LIN {X -0.105,Y -512.743,Z 1082.951,A 0.000,B 0.000,C 90.000,E1 27.206} C_DIS
LIN {X -0.246,Y -506.271,Z 1082.947,A 0.000,B 0.000,C 90.000,E1 26.488} C_DIS
LIN {X 0.235,Y -498.378,Z 1082.942,A 0.000,B 0.000,C 90.000,E1 25.591} C_DIS
LIN {X 0.081,Y -491.474,Z 1082.938,A 0.000,B 0.000,C 90.000,E1 24.899} C_DIS
LIN {X 0.101,Y -483.056,Z 1082.934,A 0.000,B 0.000,C 90.000,E1 24.079} C_DIS
LIN {X 0.080,Y -473.077,Z 1082.929,A 0.000,B 0.000,C 90.000,E1 23.153} C_DIS
LIN {X -0.074,Y -468.531,Z 1082.927,A 0.000,B 0.000,C 90.000,E1 22.770} C_DIS
LIN {X 0.200,Y -458.259,Z 1082.922,A 0.000,B 0.000,C 90.000,E1 21.844} C_DIS
LIN {X -0.133,Y -450.699,Z 1082.918,A 0.000,B 0.000,C 90.000,E1 21.227} C_DIS
LIN {X -0.068,Y -433.276,Z 1082.909,A 0.000,B 0.000,C 90.000,E1 19.631} C_DIS
LIN {X -0.013,Y -417.456,Z 1082.900,A 0.000,B 0.000,C 90.000,E1 18.000} C_DIS
LIN {X 0.024,Y -405.312,Z 1082.892,A 0.000,B 0.000,C 90.000,E1 16.567} C_DIS
LIN {X 0.104,Y -399.058,Z 1082.887,A 0.000,B 0.000,C 90.000,E1 15.717} C_DIS
LIN {X 0.077,Y -396.824,Z 1082.885,A 0.000,B 0.000,C 90.000,E1 15.371} C_DIS
LIN {X -0.054,Y -394.256,Z 1082.883,A 0.000,B 0.000,C 90.000,E1 14.898} C_DIS
LIN {X 0.015,Y -392.680,Z 1082.880,A 0.000,B 0.000,C 90.000,E1 14.356} C_DIS
LIN {X -0.009,Y -392.087,Z 1082.877,A 0.000,B 0.000,C 90.000,E1 13.828} C_DIS
LIN {X 0.012,Y -392.010,Z 1082.876,A 0.000,B 0.000,C 90.000,E1 13.647} C_DIS
LIN {X -0.076,Y -392.528,Z 1082.871,A 0.000,B 0.000,C 90.000,E1 12.771} C_DIS
LIN {X -0.071,Y -394.325,Z 1082.863,A 0.000,B 0.000,C 90.000,E1 11.366} C_DIS
LIN {X 0.118,Y -400.821,Z 1082.844,A 0.000,B 0.000,C 90.000,E1 7.814} C_DIS
LIN {X -0.026,Y -405.485,Z 1082.832,A 0.000,B 0.000,C 90.000,E1 5.739} C_DIS
LIN {X -0.062,Y -406.947,Z 1082.828,A 0.000,B 0.000,C 90.000,E1 5.049} C_DIS
LIN {X -0.086,Y -409.086,Z 1082.824,A 0.000,B 0.000,C 90.000,E1 4.359} C_DIS
LIN {X -0.078,Y -410.586,Z 1082.822,A 0.000,B 0.000,C 90.000,E1 4.012} C_DIS
LIN {X -0.092,Y -412.395,Z 1082.820,A 0.000,B 0.000,C 90.000,E1 3.669} C_DIS
LIN {X -0.098,Y -415.251,Z 1082.818,A 0.000,B 0.000,C 90.000,E1 3.326} C_DIS
LIN {X 0.044,Y -417.972,Z 1082.817,A 0.000,B 0.000,C 90.000,E1 3.037} C_DIS
LIN {X 0.077,Y -421.563,Z 1082.815,A 0.000,B 0.000,C 90.000,E1 2.751} C_DIS
LIN {X -0.121,Y -429.063,Z 1082.813,A 0.000,B 0.000,C 90.000,E1 2.293} C_DIS
LIN {X 0.017,Y -448.904,Z 1082.805,A 0.000,B 0.000,C 90.000,E1 0.974} C_DIS
LIN {X 0.000,Y -464.386,Z 1082.800,A 0.000,B 0.000,C 90.000,E1 360.000} C_DIS
LIN {X 0.157,Y -474.218,Z 1082.797,A 0.000,B 0.000,C 90.000,E1 359.370} C_DIS
LIN {X -0.054,Y -485.618,Z 1082.793,A 0.000,B 0.000,C 90.000,E1 358.682} C_DIS
LIN {X -0.189,Y -491.941,Z 1082.790,A 0.000,B 0.000,C 90.000,E1 358.282} C_DIS
LIN {X 0.157,Y -499.792,Z 1082.787,A 0.000,B 0.000,C 90.000,E1 357.707} C_DIS
LIN {X -0.201,Y -504.418,Z 1082.786,A 0.000,B 0.000,C 90.000,E1 357.421} C_DIS
LIN {X -0.122,Y -510.460,Z 1082.783,A 0.000,B 0.000,C 90.000,E1 356.963} C_DIS
LIN {X -0.140,Y -516.466,Z 1082.781,A 0.000,B 0.000,C 90.000,E1 356.502} C_DIS
LIN {X 0.074,Y -523.648,Z 1082.777,A 0.000,B 0.000,C 90.000,E1 355.869} C_DIS
LIN {X 0.106,Y -528.999,Z 1082.774,A 0.000,B 0.000,C 90.000,E1 355.355} C_DIS
LIN {X -0.259,Y -533.999,Z 1082.771,A 0.000,B 0.000,C 90.000,E1 354.894} C_DIS
LIN {X -0.088,Y -539.075,Z 1082.768,A 0.000,B 0.000,C 90.000,E1 354.318} C_DIS
LIN {X 0.248,Y -544.958,Z 1082.765,A 0.000,B 0.000,C 90.000,E1 353.571} C_DIS
LIN {X 0.066,Y -548.338,Z 1082.762,A 0.000,B 0.000,C 90.000,E1 353.166} C_DIS
LIN {X 0.008,Y -553.208,Z 1082.758,A 0.000,B 0.000,C 90.000,E1 352.470} C_DIS
LIN {X -0.083,Y -557.570,Z 1082.754,A 0.000,B 0.000,C 90.000,E1 351.781} C_DIS
LIN {X 0.189,Y -560.730,Z 1082.751,A 0.000,B 0.000,C 90.000,E1 351.197} C_DIS
LIN {X 0.248,Y -564.312,Z 1082.747,A 0.000,B 0.000,C 90.000,E1 350.500} C_DIS
LIN {X -0.221,Y -567.611,Z 1082.744,A 0.000,B 0.000,C 90.000,E1 349.859} C_DIS
LIN {X 0.031,Y -570.045,Z 1082.741,A 0.000,B 0.000,C 90.000,E1 349.285} C_DIS
LIN {X 0.226,Y -574.569,Z 1082.734,A 0.000,B 0.000,C 90.000,E1 348.173} C_DIS
LIN {X -0.288,Y -577.679,Z 1082.730,A 0.000,B 0.000,C 90.000,E1 347.409} C_DIS
LIN {X -0.208,Y -580.742,Z 1082.725,A 0.000,B 0.000,C 90.000,E1 346.589} C_DIS
LIN {X 0.182,Y -586.351,Z 1082.716,A 0.000,B 0.000,C 90.000,E1 344.936} C_DIS
LIN {X 0.028,Y -590.694,Z 1082.709,A 0.000,B 0.000,C 90.000,E1 343.614} C_DIS
LIN {X -0.219,Y -594.814,Z 1082.702,A 0.000,B 0.000,C 90.000,E1 342.308} C_DIS
LIN {X 0.070,Y -598.009,Z 1082.696,A 0.000,B 0.000,C 90.000,E1 341.221} C_DIS
LIN {X 0.019,Y -602.177,Z 1082.687,A 0.000,B 0.000,C 90.000,E1 339.645} C_DIS
LIN {X 0.127,Y -604.055,Z 1082.683,A 0.000,B 0.000,C 90.000,E1 338.847} C_DIS
LIN {X 0.191,Y -606.370,Z 1082.677,A 0.000,B 0.000,C 90.000,E1 337.794} C_DIS
LIN {X 0.236,Y -608.760,Z 1082.670,A 0.000,B 0.000,C 90.000,E1 336.485} C_DIS
LIN {X -0.194,Y -610.357,Z 1082.664,A 0.000,B 0.000,C 90.000,E1 335.485} C_DIS
LIN {X 0.240,Y -611.498,Z 1082.659,A 0.000,B 0.000,C 90.000,E1 334.665} C_DIS
LIN {X 0.073,Y -613.069,Z 1082.652,A 0.000,B 0.000,C 90.000,E1 333.384} C_DIS
LIN {X -0.015,Y -613.870,Z 1082.648,A 0.000,B 0.000,C 90.000,E1 332.615} C_DIS
LIN {X 0.168,Y -614.764,Z 1082.642,A 0.000,B 0.000,C 90.000,E1 331.563} C_DIS
LIN {X 0.066,Y -615.301,Z 1082.636,A 0.000,B 0.000,C 90.000,E1 330.539} C_DIS
LIN {X -0.268,Y -615.607,Z 1082.631,A 0.000,B 0.000,C 90.000,E1 329.537} C_DIS
LIN {X 0.252,Y -615.430,Z 1082.625,A 0.000,B 0.000,C 90.000,E1 328.456} C_DIS
LIN {X -0.077,Y -614.933,Z 1082.619,A 0.000,B 0.000,C 90.000,E1 327.454} C_DIS
LIN {X -0.085,Y -614.033,Z 1082.613,A 0.000,B 0.000,C 90.000,E1 326.421} C_DIS
LIN {X 0.189,Y -612.460,Z 1082.606,A 0.000,B 0.000,C 90.000,E1 325.102} C_DIS
LIN {X -0.146,Y -611.447,Z 1082.602,A 0.000,B 0.000,C 90.000,E1 324.356} C_DIS
LIN {X 0.224,Y -609.559,Z 1082.593,A 0.000,B 0.000,C 90.000,E1 322.763} C_DIS
LIN {X -0.293,Y -607.736,Z 1082.585,A 0.000,B 0.000,C 90.000,E1 321.251} C_DIS
LIN {X -0.082,Y -606.156,Z 1082.576,A 0.000,B 0.000,C 90.000,E1 319.666} C_DIS
LIN {X -0.097,Y -604.273,Z 1082.566,A 0.000,B 0.000,C 90.000,E1 317.838} C_DIS
LIN {X -0.049,Y -603.668,Z 1082.563,A 0.000,B 0.000,C 90.000,E1 317.310} C_DIS
LIN {X -0.209,Y -602.585,Z 1082.558,A 0.000,B 0.000,C 90.000,E1 316.539} C_DIS
LIN {X 0.060,Y -599.970,Z 1082.548,A 0.000,B 0.000,C 90.000,E1 314.676} C_DIS
LIN {X -0.152,Y -598.236,Z 1082.541,A 0.000,B 0.000,C 90.000,E1 313.380} C_DIS
LIN {X 0.246,Y -595.387,Z 1082.529,A 0.000,B 0.000,C 90.000,E1 311.229} C_DIS
LIN {X -0.018,Y -593.384,Z 1082.522,A 0.000,B 0.000,C 90.000,E1 309.930} C_DIS
LIN {X 0.169,Y -592.012,Z 1082.517,A 0.000,B 0.000,C 90.000,E1 309.116} C_DIS
LIN {X -0.074,Y -589.339,Z 1082.510,A 0.000,B 0.000,C 90.000,E1 307.810} C_DIS
LIN {X 0.108,Y -586.240,Z 1082.503,A 0.000,B 0.000,C 90.000,E1 306.457} C_DIS
LIN {X 0.020,Y -584.738,Z 1082.500,A 0.000,B 0.000,C 90.000,E1 305.931} C_DIS
LIN {X -0.134,Y -583.880,Z 1082.498,A 0.000,B 0.000,C 90.000,E1 305.678} C_DIS
LIN {X 0.233,Y -582.438,Z 1082.495,A 0.000,B 0.000,C 90.000,E1 305.105} C_DIS
LIN {X -0.223,Y -580.788,Z 1082.492,A 0.000,B 0.000,C 90.000,E1 304.612} C_DIS
LIN {X 0.115,Y -578.836,Z 1082.489,A 0.000,B 0.000,C 90.000,E1 304.040} C_DIS
LIN {X 0.114,Y -576.720,Z 1082.486,A 0.000,B 0.000,C 90.000,E1 303.499} C_DIS
LIN {X 0.013,Y -573.478,Z 1082.482,A 0.000,B 0.000,C 90.000,E1 302.832} C_DIS
LIN {X 0.013,Y -568.208,Z 1082.477,A 0.000,B 0.000,C 90.000,E1 301.878} C_DIS
LIN {X -0.079,Y -567.363,Z 1082.476,A 0.000,B 0.000,C 90.000,E1 301.750} C_DIS
LIN {X -0.063,Y -560.691,Z 1082.472,A 0.000,B 0.000,C 90.000,E1 300.924} C_DIS
LIN {X -0.157,Y -555.536,Z 1082.469,A 0.000,B 0.000,C 90.000,E1 300.384} C_DIS
LIN {X -0.123,Y -552.525,Z 1082.467,A 0.000,B 0.000,C 90.000,E1 300.129} C_DIS
LIN {X 0.055,Y -547.457,Z 1082.465,A 0.000,B 0.000,C 90.000,E1 299.617} C_DIS
LIN {X -0.277,Y -546.455,Z 1082.464,A 0.000,B 0.000,C 90.000,E1 299.539} C_DIS
LIN {X -0.028,Y -544.583,Z 1082.462,A 0.000,B 0.000,C 90.000,E1 299.205} C_DIS
LIN {X -0.152,Y -543.636,Z 1082.462,A 0.000,B 0.000,C 90.000,E1 299.077} C_DIS
LIN {X 0.205,Y -542.356,Z 1082.459,A 0.000,B 0.000,C 90.000,E1 298.615} C_DIS
LIN {X 0.076,Y -542.284,Z 1082.458,A 0.000,B 0.000,C 90.000,E1 298.487} C_DIS
LIN {X -0.150,Y -542.015,Z 1082.458,A 0.000,B 0.000,C 90.000,E1 298.359} C_DIS
LIN {X 0.069,Y -541.254,Z 1082.456,A 0.000,B 0.000,C 90.000,E1 298.052} C_DIS
LIN {X 0.063,Y -541.031,Z 1082.454,A 0.000,B 0.000,C 90.000,E1 297.769} C_DIS
LIN {X 0.149,Y -540.497,Z 1082.452,A 0.000,B 0.000,C 90.000,E1 297.334} C_DIS
LIN {X 0.019,Y -540.575,Z 1082.451,A 0.000,B 0.000,C 90.000,E1 297.206} C_DIS
LIN {X 0.000,Y -540.494,Z 1082.450,A 0.000,B 0.000,C 90.000,E1 296.924} C_DIS
LIN {X 0.219,Y -540.223,Z 1082.448,A 0.000,B 0.000,C 90.000,E1 296.616} C_DIS
LIN {X 0.061,Y -540.481,Z 1082.431,A 0.000,B 0.000,C 90.000,E1 293.590} C_DIS
LIN {X 0.215,Y -540.875,Z 1082.423,A 0.000,B 0.000,C 90.000,E1 292.153} C_DIS
LIN {X -0.105,Y -541.428,Z 1082.414,A 0.000,B 0.000,C 90.000,E1 290.482} C_DIS
LIN {X 0.126,Y -541.613,Z 1082.407,A 0.000,B 0.000,C 90.000,E1 289.322} C_DIS
LIN {X 0.183,Y -541.648,Z 1082.401,A 0.000,B 0.000,C 90.000,E1 288.181} C_DIS
LIN {X 0.015,Y -541.453,Z 1082.392,A 0.000,B 0.000,C 90.000,E1 286.496} C_DIS
LIN {X 0.134,Y -541.076,Z 1082.384,A 0.000,B 0.000,C 90.000,E1 285.064} C_DIS
LIN {X 0.104,Y -540.565,Z 1082.376,A 0.000,B 0.000,C 90.000,E1 283.647} C_DIS
LIN {X -0.055,Y -539.946,Z 1082.368,A 0.000,B 0.000,C 90.000,E1 282.243} C_DIS
LIN {X -0.219,Y -539.205,Z 1082.360,A 0.000,B 0.000,C 90.000,E1 280.838} C_DIS
LIN {X 0.233,Y -538.052,Z 1082.347,A 0.000,B 0.000,C 90.000,E1 278.511} C_DIS
LIN {X -0.089,Y -537.157,Z 1082.338,A 0.000,B 0.000,C 90.000,E1 276.834} C_DIS
LIN {X 0.042,Y -536.295,Z 1082.328,A 0.000,B 0.000,C 90.000,E1 275.106} C_DIS
LIN {X 0.112,Y -535.382,Z 1082.319,A 0.000,B 0.000,C 90.000,E1 273.383} C_DIS
LIN {X 0.154,Y -534.529,Z 1082.309,A 0.000,B 0.000,C 90.000,E1 271.661} C_DIS
LIN {X 0.147,Y -534.032,Z 1082.303,A 0.000,B 0.000,C 90.000,E1 270.516} C_DIS
LIN {X 0.126,Y -533.069,Z 1082.293,A 0.000,B 0.000,C 90.000,E1 268.797} C_DIS
LIN {X 0.092,Y -532.058,Z 1082.284,A 0.000,B 0.000,C 90.000,E1 267.078} C_DIS
LIN {X 0.100,Y -531.420,Z 1082.277,A 0.000,B 0.000,C 90.000,E1 265.927} C_DIS
LIN {X 0.058,Y -530.119,Z 1082.268,A 0.000,B 0.000,C 90.000,E1 264.204} C_DIS
LIN {X 0.066,Y -528.841,Z 1082.260,A 0.000,B 0.000,C 90.000,E1 262.761} C_DIS
LIN {X 0.093,Y -526.698,Z 1082.249,A 0.000,B 0.000,C 90.000,E1 260.735} C_DIS
LIN {X 0.107,Y -525.157,Z 1082.241,A 0.000,B 0.000,C 90.000,E1 259.285} C_DIS
LIN {X 0.184,Y -523.654,Z 1082.233,A 0.000,B 0.000,C 90.000,E1 257.825} C_DIS
LIN {X -0.156,Y -521.929,Z 1082.223,A 0.000,B 0.000,C 90.000,E1 256.117} C_DIS
LIN {X 0.104,Y -520.178,Z 1082.213,A 0.000,B 0.000,C 90.000,E1 254.338} C_DIS
LIN {X -0.029,Y -518.351,Z 1082.203,A 0.000,B 0.000,C 90.000,E1 252.598} C_DIS
LIN {X -0.167,Y -516.791,Z 1082.195,A 0.000,B 0.000,C 90.000,E1 251.148} C_DIS
LIN {X 0.143,Y -515.178,Z 1082.187,A 0.000,B 0.000,C 90.000,E1 249.645} C_DIS
LIN {X -0.057,Y -512.961,Z 1082.177,A 0.000,B 0.000,C 90.000,E1 247.901} C_DIS
LIN {X 0.180,Y -510.485,Z 1082.167,A 0.000,B 0.000,C 90.000,E1 246.102} C_DIS
LIN {X 0.141,Y -508.671,Z 1082.161,A 0.000,B 0.000,C 90.000,E1 244.921} C_DIS
LIN {X -0.173,Y -506.824,Z 1082.154,A 0.000,B 0.000,C 90.000,E1 243.768} C_DIS
LIN {X -0.139,Y -505.365,Z 1082.149,A 0.000,B 0.000,C 90.000,E1 242.871} C_DIS
LIN {X -0.193,Y -502.859,Z 1082.141,A 0.000,B 0.000,C 90.000,E1 241.385} C_DIS
LIN {X 0.237,Y -499.776,Z 1082.131,A 0.000,B 0.000,C 90.000,E1 239.537} C_DIS
LIN {X -0.257,Y -496.507,Z 1082.121,A 0.000,B 0.000,C 90.000,E1 237.788} C_DIS
LIN {X 0.131,Y -493.104,Z 1082.111,A 0.000,B 0.000,C 90.000,E1 235.928} C_DIS
LIN {X 0.189,Y -490.141,Z 1082.102,A 0.000,B 0.000,C 90.000,E1 234.402} C_DIS
LIN {X -0.213,Y -487.095,Z 1082.094,A 0.000,B 0.000,C 90.000,E1 232.924} C_DIS
LIN {X 0.118,Y -483.221,Z 1082.084,A 0.000,B 0.000,C 90.000,E1 231.045} C_DIS
LIN {X -0.200,Y -479.911,Z 1082.075,A 0.000,B 0.000,C 90.000,E1 229.542} C_DIS
LIN {X 0.094,Y -474.844,Z 1082.061,A 0.000,B 0.000,C 90.000,E1 227.025} C_DIS
LIN {X 0.103,Y -470.752,Z 1082.049,A 0.000,B 0.000,C 90.000,E1 224.838} C_DIS
LIN {X -0.070,Y -467.249,Z 1082.039,A 0.000,B 0.000,C 90.000,E1 222.975} C_DIS
LIN {X 0.166,Y -465.471,Z 1082.033,A 0.000,B 0.000,C 90.000,E1 222.000} C_DIS
LIN {X -0.017,Y -461.185,Z 1082.021,A 0.000,B 0.000,C 90.000,E1 219.806} C_DIS
LIN {X -0.082,Y -458.171,Z 1082.012,A 0.000,B 0.000,C 90.000,E1 218.222} C_DIS
LIN {X -0.048,Y -454.475,Z 1082.002,A 0.000,B 0.000,C 90.000,E1 216.297} C_DIS
LIN {X -0.159,Y -452.026,Z 1081.995,A 0.000,B 0.000,C 90.000,E1 215.025} C_DIS
LIN {X -0.005,Y -447.147,Z 1081.980,A 0.000,B 0.000,C 90.000,E1 212.418} C_DIS
LIN {X 0.018,Y -443.605,Z 1081.969,A 0.000,B 0.000,C 90.000,E1 210.463} C_DIS
LIN {X 0.112,Y -440.141,Z 1081.958,A 0.000,B 0.000,C 90.000,E1 208.487} C_DIS
LIN {X 0.148,Y -435.672,Z 1081.944,A 0.000,B 0.000,C 90.000,E1 205.848} C_DIS
LIN {X 0.214,Y -433.861,Z 1081.936,A 0.000,B 0.000,C 90.000,E1 204.515} C_DIS
LIN {X -0.099,Y -430.329,Z 1081.922,A 0.000,B 0.000,C 90.000,E1 201.897} C_DIS
LIN {X -0.243,Y -428.987,Z 1081.912,A 0.000,B 0.000,C 90.000,E1 200.248} C_DIS
LIN {X -0.227,Y -428.850,Z 1081.909,A 0.000,B 0.000,C 90.000,E1 199.577} C_DIS
LIN {X -0.213,Y -429.007,Z 1081.905,A 0.000,B 0.000,C 90.000,E1 198.906} C_DIS
LIN {X 0.207,Y -429.520,Z 1081.901,A 0.000,B 0.000,C 90.000,E1 198.181} C_DIS
LIN {X 0.221,Y -430.422,Z 1081.897,A 0.000,B 0.000,C 90.000,E1 197.511} C_DIS
LIN {X 0.111,Y -431.796,Z 1081.894,A 0.000,B 0.000,C 90.000,E1 196.858} C_DIS
LIN {X -0.085,Y -432.640,Z 1081.892,A 0.000,B 0.000,C 90.000,E1 196.551} C_DIS
LIN {X -0.069,Y -435.929,Z 1081.886,A 0.000,B 0.000,C 90.000,E1 195.552} C_DIS
LIN {X 0.107,Y -443.669,Z 1081.876,A 0.000,B 0.000,C 90.000,E1 193.716} C_DIS
LIN {X 0.166,Y -450.524,Z 1081.868,A 0.000,B 0.000,C 90.000,E1 192.243} C_DIS
LIN {X -0.068,Y -457.822,Z 1081.860,A 0.000,B 0.000,C 90.000,E1 190.838} C_DIS
LIN {X 0.113,Y -467.048,Z 1081.851,A 0.000,B 0.000,C 90.000,E1 189.095} C_DIS
LIN {X 0.063,Y -475.533,Z 1081.842,A 0.000,B 0.000,C 90.000,E1 187.530} C_DIS
LIN {X -0.011,Y -480.533,Z 1081.837,A 0.000,B 0.000,C 90.000,E1 186.606} C_DIS
LIN {X 0.116,Y -486.113,Z 1081.831,A 0.000,B 0.000,C 90.000,E1 185.511} C_DIS
LIN {X -0.009,Y -492.414,Z 1081.824,A 0.000,B 0.000,C 90.000,E1 184.302} C_DIS
LIN {X 0.129,Y -499.320,Z 1081.816,A 0.000,B 0.000,C 90.000,E1 182.922} C_DIS
LIN {X -0.053,Y -504.614,Z 1081.811,A 0.000,B 0.000,C 90.000,E1 181.892} C_DIS
LIN {X -0.244,Y -511.387,Z 1081.803,A 0.000,B 0.000,C 90.000,E1 180.573} C_DIS
LIN {X -0.170,Y -520.402,Z 1081.793,A 0.000,B 0.000,C 90.000,E1 178.797} C_DIS
LIN {X 0.145,Y -527.773,Z 1081.785,A 0.000,B 0.000,C 90.000,E1 177.306} C_DIS
LIN {X -0.194,Y -534.352,Z 1081.778,A 0.000,B 0.000,C 90.000,E1 176.045} C_DIS
LIN {X -0.124,Y -541.601,Z 1081.770,A 0.000,B 0.000,C 90.000,E1 174.609} C_DIS
LIN {X 0.110,Y -547.347,Z 1081.764,A 0.000,B 0.000,C 90.000,E1 173.451} C_DIS
LIN {X -0.017,Y -555.815,Z 1081.754,A 0.000,B 0.000,C 90.000,E1 171.781} C_DIS
LIN {X 0.281,Y -561.957,Z 1081.747,A 0.000,B 0.000,C 90.000,E1 170.500} C_DIS
LIN {X -0.110,Y -568.683,Z 1081.740,A 0.000,B 0.000,C 90.000,E1 169.162} C_DIS
LIN {X 0.282,Y -575.057,Z 1081.732,A 0.000,B 0.000,C 90.000,E1 167.757} C_DIS
LIN {X -0.017,Y -581.736,Z 1081.724,A 0.000,B 0.000,C 90.000,E1 166.297} C_DIS
LIN {X -0.168,Y -587.013,Z 1081.717,A 0.000,B 0.000,C 90.000,E1 165.102} C_DIS
LIN {X 0.102,Y -592.400,Z 1081.710,A 0.000,B 0.000,C 90.000,E1 163.740} C_DIS
LIN {X -0.081,Y -595.449,Z 1081.705,A 0.000,B 0.000,C 90.000,E1 162.960} C_DIS
LIN {X 0.224,Y -599.333,Z 1081.699,A 0.000,B 0.000,C 90.000,E1 161.873} C_DIS
LIN {X 0.111,Y -602.132,Z 1081.695,A 0.000,B 0.000,C 90.000,E1 161.094} C_DIS
LIN {X -0.135,Y -606.421,Z 1081.688,A 0.000,B 0.000,C 90.000,E1 159.806} C_DIS
LIN {X 0.265,Y -610.476,Z 1081.681,A 0.000,B 0.000,C 90.000,E1 158.465} C_DIS
LIN {X 0.154,Y -614.298,Z 1081.673,A 0.000,B 0.000,C 90.000,E1 157.177} C_DIS
LIN {X -0.227,Y -617.908,Z 1081.666,A 0.000,B 0.000,C 90.000,E1 155.921} C_DIS
LIN {X 0.006,Y -621.912,Z 1081.658,A 0.000,B 0.000,C 90.000,E1 154.357} C_DIS
LIN {X 0.013,Y -625.143,Z 1081.651,A 0.000,B 0.000,C 90.000,E1 153.076} C_DIS
LIN {X 0.368,Y -628.222,Z 1081.643,A 0.000,B 0.000,C 90.000,E1 151.769} C_DIS
LIN {X -0.076,Y -631.141,Z 1081.636,A 0.000,B 0.000,C 90.000,E1 150.539} C_DIS
LIN {X 0.187,Y -634.472,Z 1081.628,A 0.000,B 0.000,C 90.000,E1 148.997} C_DIS
LIN {X -0.013,Y -637.709,Z 1081.620,A 0.000,B 0.000,C 90.000,E1 147.502} C_DIS
LIN {X -0.114,Y -641.275,Z 1081.610,A 0.000,B 0.000,C 90.000,E1 145.754} C_DIS
LIN {X 0.048,Y -644.710,Z 1081.600,A 0.000,B 0.000,C 90.000,E1 143.989} C_DIS
LIN {X 0.252,Y -647.511,Z 1081.592,A 0.000,B 0.000,C 90.000,E1 142.477} C_DIS
LIN {X 0.078,Y -649.950,Z 1081.585,A 0.000,B 0.000,C 90.000,E1 141.251} C_DIS
LIN {X -0.187,Y -653.393,Z 1081.575,A 0.000,B 0.000,C 90.000,E1 139.542} C_DIS
LIN {X 0.088,Y -656.414,Z 1081.567,A 0.000,B 0.000,C 90.000,E1 138.038} C_DIS
LIN {X 0.306,Y -661.064,Z 1081.555,A 0.000,B 0.000,C 90.000,E1 135.810} C_DIS
LIN {X 0.215,Y -665.116,Z 1081.545,A 0.000,B 0.000,C 90.000,E1 134.109} C_DIS
LIN {X -0.248,Y -670.050,Z 1081.534,A 0.000,B 0.000,C 90.000,E1 132.204} C_DIS
LIN {X 0.385,Y -674.371,Z 1081.525,A 0.000,B 0.000,C 90.000,E1 130.458} C_DIS
LIN {X 0.140,Y -678.018,Z 1081.517,A 0.000,B 0.000,C 90.000,E1 129.036} C_DIS
LIN {X -0.293,Y -682.977,Z 1081.506,A 0.000,B 0.000,C 90.000,E1 127.156} C_DIS
LIN {X 0.113,Y -686.067,Z 1081.500,A 0.000,B 0.000,C 90.000,E1 125.931} C_DIS
LIN {X -0.204,Y -689.531,Z 1081.492,A 0.000,B 0.000,C 90.000,E1 124.532} C_DIS
LIN {X -0.241,Y -693.558,Z 1081.483,A 0.000,B 0.000,C 90.000,E1 122.880} C_DIS
LIN {X -0.218,Y -696.953,Z 1081.475,A 0.000,B 0.000,C 90.000,E1 121.465} C_DIS
LIN {X -0.050,Y -699.009,Z 1081.469,A 0.000,B 0.000,C 90.000,E1 120.512} C_DIS
LIN {X 0.128,Y -700.324,Z 1081.466,A 0.000,B 0.000,C 90.000,E1 119.795} C_DIS
LIN {X 0.053,Y -701.043,Z 1081.463,A 0.000,B 0.000,C 90.000,E1 119.333} C_DIS
LIN {X 0.188,Y -702.361,Z 1081.457,A 0.000,B 0.000,C 90.000,E1 118.153} C_DIS
LIN {X 0.298,Y -703.666,Z 1081.449,A 0.000,B 0.000,C 90.000,E1 116.744} C_DIS
LIN {X 0.149,Y -704.730,Z 1081.442,A 0.000,B 0.000,C 90.000,E1 115.591} C_DIS
LIN {X -0.216,Y -705.058,Z 1081.440,A 0.000,B 0.000,C 90.000,E1 115.155} C_DIS
LIN {X 0.360,Y -705.140,Z 1081.437,A 0.000,B 0.000,C 90.000,E1 114.643} C_DIS
LIN {X 0.002,Y -704.721,Z 1081.435,A 0.000,B 0.000,C 90.000,E1 114.207} C_DIS
LIN {X 0.287,Y -704.411,Z 1081.433,A 0.000,B 0.000,C 90.000,E1 113.951} C_DIS
LIN {X -0.074,Y -702.806,Z 1081.431,A 0.000,B 0.000,C 90.000,E1 113.515} C_DIS
LIN {X 0.204,Y -701.746,Z 1081.429,A 0.000,B 0.000,C 90.000,E1 113.259} C_DIS
LIN {X -0.173,Y -698.154,Z 1081.427,A 0.000,B 0.000,C 90.000,E1 112.823} C_DIS
LIN {X -0.044,Y -697.056,Z 1081.426,A 0.000,B 0.000,C 90.000,E1 112.695} C_DIS
LIN {X -0.182,Y -695.384,Z 1081.425,A 0.000,B 0.000,C 90.000,E1 112.589} C_DIS
LIN {X 0.363,Y -687.730,Z 1081.424,A 0.000,B 0.000,C 90.000,E1 112.206} C_DIS
LIN {X 0.141,Y -685.814,Z 1081.423,A 0.000,B 0.000,C 90.000,E1 112.153} C_DIS
LIN {X -0.285,Y -684.330,Z 1081.423,A 0.000,B 0.000,C 90.000,E1 112.153} C_DIS
LIN {X -0.082,Y -675.933,Z 1081.422,A 0.000,B 0.000,C 90.000,E1 112.025} C_DIS
LIN {X -0.121,Y -605.703,Z 1081.422,A 0.000,B 0.000,C 90.000,E1 112.025} C_DIS
LIN {X -0.017,Y -601.930,Z 1081.421,A 0.000,B 0.000,C 90.000,E1 111.844} C_DIS
LIN {X 0.141,Y -596.452,Z 1081.419,A 0.000,B 0.000,C 90.000,E1 111.482} C_DIS
LIN {X 0.237,Y -587.291,Z 1081.415,A 0.000,B 0.000,C 90.000,E1 110.737} C_DIS
LIN {X -0.108,Y -578.950,Z 1081.411,A 0.000,B 0.000,C 90.000,E1 110.066} C_DIS
LIN {X 0.022,Y -574.660,Z 1081.410,A 0.000,B 0.000,C 90.000,E1 109.704} C_DIS
LIN {X -0.127,Y -568.620,Z 1081.407,A 0.000,B 0.000,C 90.000,E1 109.268} C_DIS
LIN {X 0.186,Y -560.275,Z 1081.404,A 0.000,B 0.000,C 90.000,E1 108.725} C_DIS
LIN {X 0.113,Y -553.840,Z 1081.402,A 0.000,B 0.000,C 90.000,E1 108.362} C_DIS
LIN {X 0.190,Y -549.451,Z 1081.401,A 0.000,B 0.000,C 90.000,E1 108.055} C_DIS
LIN {X -0.059,Y -547.800,Z 1081.399,A 0.000,B 0.000,C 90.000,E1 107.873} C_DIS
LIN {X -0.090,Y -547.793,Z 1081.399,A 0.000,B 0.000,C 90.000,E1 107.873} C_DIS
LIN {X -0.214,Y -547.542,Z 1081.398,A 0.000,B 0.000,C 90.000,E1 107.692} C_DIS
LIN {X 0.214,Y -547.463,Z 1081.397,A 0.000,B 0.000,C 90.000,E1 107.457} C_DIS
LIN {X 0.053,Y -548.752,Z 1081.385,A 0.000,B 0.000,C 90.000,E1 105.300} C_DIS
LIN {X -0.155,Y -550.211,Z 1081.374,A 0.000,B 0.000,C 90.000,E1 103.355} C_DIS
LIN {X -0.132,Y -551.386,Z 1081.366,A 0.000,B 0.000,C 90.000,E1 101.951} C_DIS
LIN {X 0.034,Y -553.009,Z 1081.357,A 0.000,B 0.000,C 90.000,E1 100.254} C_DIS
LIN {X 0.253,Y -555.156,Z 1081.346,A 0.000,B 0.000,C 90.000,E1 98.276} C_DIS
LIN {X -0.188,Y -557.299,Z 1081.335,A 0.000,B 0.000,C 90.000,E1 96.372} C_DIS
LIN {X 0.200,Y -558.463,Z 1081.329,A 0.000,B 0.000,C 90.000,E1 95.220} C_DIS
LIN {X 0.127,Y -559.603,Z 1081.321,A 0.000,B 0.000,C 90.000,E1 93.841} C_DIS
LIN {X 0.038,Y -560.409,Z 1081.314,A 0.000,B 0.000,C 90.000,E1 92.465} C_DIS
LIN {X -0.036,Y -561.180,Z 1081.306,A 0.000,B 0.000,C 90.000,E1 91.088} C_DIS
LIN {X -0.109,Y -561.733,Z 1081.298,A 0.000,B 0.000,C 90.000,E1 89.714} C_DIS
LIN {X -0.177,Y -562.314,Z 1081.291,A 0.000,B 0.000,C 90.000,E1 88.339} C_DIS
LIN {X -0.222,Y -562.876,Z 1081.283,A 0.000,B 0.000,C 90.000,E1 86.963} C_DIS
LIN {X -0.223,Y -563.413,Z 1081.275,A 0.000,B 0.000,C 90.000,E1 85.584} C_DIS
LIN {X 0.032,Y -564.055,Z 1081.265,A 0.000,B 0.000,C 90.000,E1 83.628} C_DIS
LIN {X 0.114,Y -564.461,Z 1081.257,A 0.000,B 0.000,C 90.000,E1 82.243} C_DIS
LIN {X -0.197,Y -565.027,Z 1081.248,A 0.000,B 0.000,C 90.000,E1 80.622} C_DIS
LIN {X -0.240,Y -565.854,Z 1081.237,A 0.000,B 0.000,C 90.000,E1 78.701} C_DIS
LIN {X -0.231,Y -567.086,Z 1081.223,A 0.000,B 0.000,C 90.000,E1 76.228} C_DIS
LIN {X -0.033,Y -568.668,Z 1081.210,A 0.000,B 0.000,C 90.000,E1 73.740} C_DIS
LIN {X 0.052,Y -569.753,Z 1081.202,A 0.000,B 0.000,C 90.000,E1 72.362} C_DIS
LIN {X -0.040,Y -571.098,Z 1081.193,A 0.000,B 0.000,C 90.000,E1 70.732} C_DIS
LIN {X -0.273,Y -572.254,Z 1081.185,A 0.000,B 0.000,C 90.000,E1 69.390} C_DIS
LIN {X -0.299,Y -573.850,Z 1081.175,A 0.000,B 0.000,C 90.000,E1 67.486} C_DIS
LIN {X 0.107,Y -574.709,Z 1081.169,A 0.000,B 0.000,C 90.000,E1 66.357} C_DIS
LIN {X -0.149,Y -575.729,Z 1081.161,A 0.000,B 0.000,C 90.000,E1 65.025} C_DIS
LIN {X -0.015,Y -576.717,Z 1081.152,A 0.000,B 0.000,C 90.000,E1 63.384} C_DIS
LIN {X 0.021,Y -577.566,Z 1081.145,A 0.000,B 0.000,C 90.000,E1 62.025} C_DIS
LIN {X -0.078,Y -578.550,Z 1081.136,A 0.000,B 0.000,C 90.000,E1 60.411} C_DIS
LIN {X -0.089,Y -579.350,Z 1081.127,A 0.000,B 0.000,C 90.000,E1 58.791} C_DIS
LIN {X -0.235,Y -579.780,Z 1081.122,A 0.000,B 0.000,C 90.000,E1 57.995} C_DIS
LIN {X -0.061,Y -580.395,Z 1081.115,A 0.000,B 0.000,C 90.000,E1 56.628} C_DIS
LIN {X 0.289,Y -581.126,Z 1081.106,A 0.000,B 0.000,C 90.000,E1 54.975} C_DIS
LIN {X 0.166,Y -581.474,Z 1081.100,A 0.000,B 0.000,C 90.000,E1 53.909} C_DIS
LIN {X 0.048,Y -581.751,Z 1081.094,A 0.000,B 0.000,C 90.000,E1 52.844} C_DIS
LIN {X -0.073,Y -581.911,Z 1081.088,A 0.000,B 0.000,C 90.000,E1 51.778} C_DIS
LIN {X -0.289,Y -581.807,Z 1081.082,A 0.000,B 0.000,C 90.000,E1 50.723} C_DIS
LIN {X -0.161,Y -581.366,Z 1081.073,A 0.000,B 0.000,C 90.000,E1 49.094} C_DIS
LIN {X 0.279,Y -581.067,Z 1081.068,A 0.000,B 0.000,C 90.000,E1 48.243} C_DIS
LIN {X 0.175,Y -580.446,Z 1081.061,A 0.000,B 0.000,C 90.000,E1 46.905} C_DIS
LIN {X 0.334,Y -579.821,Z 1081.055,A 0.000,B 0.000,C 90.000,E1 45.810} C_DIS
LIN {X 0.067,Y -578.929,Z 1081.049,A 0.000,B 0.000,C 90.000,E1 44.757} C_DIS
LIN {X -0.214,Y -577.841,Z 1081.043,A 0.000,B 0.000,C 90.000,E1 43.704} C_DIS
LIN {X 0.047,Y -576.099,Z 1081.035,A 0.000,B 0.000,C 90.000,E1 42.324} C_DIS
LIN {X 0.143,Y -574.517,Z 1081.029,A 0.000,B 0.000,C 90.000,E1 41.229} C_DIS
LIN {X -0.166,Y -572.546,Z 1081.023,A 0.000,B 0.000,C 90.000,E1 40.172} C_DIS
LIN {X -0.061,Y -570.343,Z 1081.017,A 0.000,B 0.000,C 90.000,E1 39.072} C_DIS
LIN {X -0.111,Y -568.443,Z 1081.013,A 0.000,B 0.000,C 90.000,E1 38.257} C_DIS
LIN {X -0.308,Y -567.085,Z 1081.010,A 0.000,B 0.000,C 90.000,E1 37.729} C_DIS
LIN {X 0.049,Y -564.659,Z 1081.005,A 0.000,B 0.000,C 90.000,E1 36.870} C_DIS
LIN {X 0.379,Y -562.046,Z 1081.000,A 0.000,B 0.000,C 90.000,E1 36.011} C_DIS
LIN {X -0.202,Y -560.018,Z 1080.997,A 0.000,B 0.000,C 90.000,E1 35.518} C_DIS
LIN {X -0.016,Y -557.782,Z 1080.994,A 0.000,B 0.000,C 90.000,E1 34.945} C_DIS
LIN {X -0.205,Y -553.683,Z 1080.989,A 0.000,B 0.000,C 90.000,E1 33.992} C_DIS
LIN {X -0.194,Y -550.436,Z 1080.985,A 0.000,B 0.000,C 90.000,E1 33.293} C_DIS
LIN {X -0.014,Y -545.495,Z 1080.979,A 0.000,B 0.000,C 90.000,E1 32.291} C_DIS
LIN {X -0.219,Y -540.953,Z 1080.975,A 0.000,B 0.000,C 90.000,E1 31.465} C_DIS
LIN {X 0.123,Y -536.922,Z 1080.971,A 0.000,B 0.000,C 90.000,E1 30.718} C_DIS
LIN {X 0.006,Y -531.747,Z 1080.966,A 0.000,B 0.000,C 90.000,E1 29.873} C_DIS
LIN {X -0.008,Y -526.832,Z 1080.962,A 0.000,B 0.000,C 90.000,E1 29.155} C_DIS
LIN {X 0.092,Y -522.686,Z 1080.959,A 0.000,B 0.000,C 90.000,E1 28.565} C_DIS
LIN {X 0.160,Y -518.207,Z 1080.956,A 0.000,B 0.000,C 90.000,E1 27.975} C_DIS
LIN {X -0.094,Y -514.710,Z 1080.953,A 0.000,B 0.000,C 90.000,E1 27.564} C_DIS
LIN {X 0.133,Y -509.773,Z 1080.950,A 0.000,B 0.000,C 90.000,E1 26.950} C_DIS
LIN {X 0.187,Y -504.534,Z 1080.947,A 0.000,B 0.000,C 90.000,E1 26.360} C_DIS
LIN {X -0.249,Y -495.063,Z 1080.941,A 0.000,B 0.000,C 90.000,E1 25.412} C_DIS
LIN {X 0.261,Y -486.695,Z 1080.936,A 0.000,B 0.000,C 90.000,E1 24.515} C_DIS
LIN {X -0.102,Y -479.473,Z 1080.933,A 0.000,B 0.000,C 90.000,E1 23.875} C_DIS
LIN {X -0.129,Y -472.261,Z 1080.929,A 0.000,B 0.000,C 90.000,E1 23.206} C_DIS
LIN {X 0.102,Y -460.448,Z 1080.923,A 0.000,B 0.000,C 90.000,E1 22.153} C_DIS
LIN {X 0.220,Y -448.498,Z 1080.917,A 0.000,B 0.000,C 90.000,E1 21.099} C_DIS
LIN {X 0.067,Y -431.039,Z 1080.908,A 0.000,B 0.000,C 90.000,E1 19.504} C_DIS
LIN {X -0.082,Y -416.825,Z 1080.900,A 0.000,B 0.000,C 90.000,E1 18.055} C_DIS
LIN {X 0.058,Y -404.831,Z 1080.892,A 0.000,B 0.000,C 90.000,E1 16.622} C_DIS
LIN {X -0.182,Y -398.767,Z 1080.888,A 0.000,B 0.000,C 90.000,E1 15.843} C_DIS
LIN {X 0.181,Y -396.812,Z 1080.886,A 0.000,B 0.000,C 90.000,E1 15.481} C_DIS
LIN {X -0.148,Y -393.707,Z 1080.883,A 0.000,B 0.000,C 90.000,E1 14.898} C_DIS
LIN {X 0.086,Y -392.293,Z 1080.879,A 0.000,B 0.000,C 90.000,E1 14.245} C_DIS
LIN {X 0.060,Y -391.908,Z 1080.876,A 0.000,B 0.000,C 90.000,E1 13.716} C_DIS
LIN {X 0.140,Y -392.581,Z 1080.871,A 0.000,B 0.000,C 90.000,E1 12.771} C_DIS
LIN {X 0.085,Y -394.997,Z 1080.861,A 0.000,B 0.000,C 90.000,E1 11.007} C_DIS
LIN {X 0.175,Y -401.576,Z 1080.842,A 0.000,B 0.000,C 90.000,E1 7.473} C_DIS
LIN {X 0.099,Y -405.478,Z 1080.832,A 0.000,B 0.000,C 90.000,E1 5.739} C_DIS
LIN {X 0.064,Y -406.919,Z 1080.828,A 0.000,B 0.000,C 90.000,E1 5.049} C_DIS
LIN {X 0.044,Y -408.974,Z 1080.824,A 0.000,B 0.000,C 90.000,E1 4.359} C_DIS
LIN {X 0.045,Y -411.244,Z 1080.821,A 0.000,B 0.000,C 90.000,E1 3.841} C_DIS
LIN {X -0.170,Y -412.541,Z 1080.820,A 0.000,B 0.000,C 90.000,E1 3.612} C_DIS
LIN {X 0.080,Y -416.093,Z 1080.818,A 0.000,B 0.000,C 90.000,E1 3.154} C_DIS
LIN {X 0.150,Y -417.820,Z 1080.817,A 0.000,B 0.000,C 90.000,E1 2.980} C_DIS
LIN {X 0.188,Y -421.445,Z 1080.815,A 0.000,B 0.000,C 90.000,E1 2.694} C_DIS
LIN {X -0.112,Y -429.154,Z 1080.812,A 0.000,B 0.000,C 90.000,E1 2.236} C_DIS
LIN {X -0.108,Y -453.804,Z 1080.803,A 0.000,B 0.000,C 90.000,E1 0.630} C_DIS
LIN {X 0.047,Y -471.866,Z 1080.797,A 0.000,B 0.000,C 90.000,E1 359.484} C_DIS
LIN {X -0.030,Y -484.862,Z 1080.793,A 0.000,B 0.000,C 90.000,E1 358.682} C_DIS
LIN {X -0.014,Y -492.704,Z 1080.790,A 0.000,B 0.000,C 90.000,E1 358.165} C_DIS
LIN {X -0.060,Y -500.385,Z 1080.787,A 0.000,B 0.000,C 90.000,E1 357.650} C_DIS
LIN {X 0.101,Y -506.506,Z 1080.785,A 0.000,B 0.000,C 90.000,E1 357.192} C_DIS
LIN {X 0.126,Y -512.595,Z 1080.782,A 0.000,B 0.000,C 90.000,E1 356.731} C_DIS
LIN {X 0.078,Y -517.106,Z 1080.780,A 0.000,B 0.000,C 90.000,E1 356.388} C_DIS
LIN {X -0.221,Y -524.244,Z 1080.777,A 0.000,B 0.000,C 90.000,E1 355.812} C_DIS
LIN {X 0.202,Y -530.964,Z 1080.773,A 0.000,B 0.000,C 90.000,E1 355.122} C_DIS
LIN {X 0.028,Y -534.498,Z 1080.771,A 0.000,B 0.000,C 90.000,E1 354.780} C_DIS
LIN {X -0.034,Y -538.335,Z 1080.769,A 0.000,B 0.000,C 90.000,E1 354.375} C_DIS
LIN {X -0.189,Y -544.279,Z 1080.765,A 0.000,B 0.000,C 90.000,E1 353.685} C_DIS
LIN {X -0.094,Y -548.798,Z 1080.762,A 0.000,B 0.000,C 90.000,E1 353.109} C_DIS
LIN {X -0.152,Y -553.633,Z 1080.758,A 0.000,B 0.000,C 90.000,E1 352.413} C_DIS
LIN {X -0.239,Y -557.971,Z 1080.754,A 0.000,B 0.000,C 90.000,E1 351.724} C_DIS
LIN {X 0.035,Y -561.134,Z 1080.751,A 0.000,B 0.000,C 90.000,E1 351.141} C_DIS
LIN {X -0.150,Y -565.385,Z 1080.746,A 0.000,B 0.000,C 90.000,E1 350.330} C_DIS
LIN {X 0.187,Y -568.011,Z 1080.743,A 0.000,B 0.000,C 90.000,E1 349.746} C_DIS
LIN {X 0.122,Y -569.873,Z 1080.741,A 0.000,B 0.000,C 90.000,E1 349.342} C_DIS
LIN {X -0.243,Y -574.450,Z 1080.735,A 0.000,B 0.000,C 90.000,E1 348.285} C_DIS
LIN {X -0.193,Y -577.618,Z 1080.730,A 0.000,B 0.000,C 90.000,E1 347.465} C_DIS
LIN {X 0.110,Y -581.674,Z 1080.724,A 0.000,B 0.000,C 90.000,E1 346.353} C_DIS
LIN {X 0.283,Y -586.359,Z 1080.717,A 0.000,B 0.000,C 90.000,E1 344.991} C_DIS
LIN {X 0.284,Y -589.898,Z 1080.711,A 0.000,B 0.000,C 90.000,E1 343.921} C_DIS
LIN {X 0.199,Y -594.119,Z 1080.703,A 0.000,B 0.000,C 90.000,E1 342.598} C_DIS
LIN {X -0.269,Y -597.400,Z 1080.698,A 0.000,B 0.000,C 90.000,E1 341.583} C_DIS
LIN {X -0.212,Y -599.615,Z 1080.693,A 0.000,B 0.000,C 90.000,E1 340.786} C_DIS
LIN {X 0.064,Y -603.063,Z 1080.686,A 0.000,B 0.000,C 90.000,E1 339.444} C_DIS
LIN {X 0.189,Y -604.919,Z 1080.682,A 0.000,B 0.000,C 90.000,E1 338.646} C_DIS
LIN {X 0.042,Y -607.170,Z 1080.676,A 0.000,B 0.000,C 90.000,E1 337.614} C_DIS
LIN {X 0.147,Y -609.138,Z 1080.670,A 0.000,B 0.000,C 90.000,E1 336.561} C_DIS
LIN {X -0.032,Y -610.789,Z 1080.664,A 0.000,B 0.000,C 90.000,E1 335.537} C_DIS
LIN {X 0.114,Y -612.279,Z 1080.658,A 0.000,B 0.000,C 90.000,E1 334.485} C_DIS
LIN {X -0.047,Y -613.853,Z 1080.651,A 0.000,B 0.000,C 90.000,E1 333.204} C_DIS
LIN {X 0.154,Y -614.652,Z 1080.647,A 0.000,B 0.000,C 90.000,E1 332.410} C_DIS
LIN {X 0.057,Y -615.539,Z 1080.641,A 0.000,B 0.000,C 90.000,E1 331.385} C_DIS
LIN {X 0.263,Y -616.081,Z 1080.635,A 0.000,B 0.000,C 90.000,E1 330.333} C_DIS
LIN {X -0.032,Y -616.323,Z 1080.631,A 0.000,B 0.000,C 90.000,E1 329.587} C_DIS
LIN {X 0.183,Y -616.289,Z 1080.625,A 0.000,B 0.000,C 90.000,E1 328.535} C_DIS
LIN {X 0.157,Y -615.760,Z 1080.618,A 0.000,B 0.000,C 90.000,E1 327.248} C_DIS
LIN {X 0.162,Y -614.913,Z 1080.612,A 0.000,B 0.000,C 90.000,E1 326.215} C_DIS
LIN {X -0.405,Y -613.452,Z 1080.605,A 0.000,B 0.000,C 90.000,E1 324.975} C_DIS
LIN {X -0.064,Y -611.380,Z 1080.595,A 0.000,B 0.000,C 90.000,E1 323.130} C_DIS
LIN {X -0.099,Y -608.478,Z 1080.579,A 0.000,B 0.000,C 90.000,E1 320.275} C_DIS
LIN {X 0.325,Y -607.228,Z 1080.572,A 0.000,B 0.000,C 90.000,E1 318.933} C_DIS
LIN {X 0.265,Y -606.080,Z 1080.565,A 0.000,B 0.000,C 90.000,E1 317.634} C_DIS
LIN {X -0.068,Y -604.875,Z 1080.559,A 0.000,B 0.000,C 90.000,E1 316.620} C_DIS
LIN {X -0.196,Y -603.127,Z 1080.552,A 0.000,B 0.000,C 90.000,E1 315.324} C_DIS
LIN {X 0.032,Y -602.742,Z 1080.550,A 0.000,B 0.000,C 90.000,E1 315.040} C_DIS
LIN {X 0.258,Y -602.535,Z 1080.549,A 0.000,B 0.000,C 90.000,E1 314.757} C_DIS
LIN {X -0.147,Y -601.777,Z 1080.546,A 0.000,B 0.000,C 90.000,E1 314.271} C_DIS
LIN {X -0.119,Y -600.678,Z 1080.540,A 0.000,B 0.000,C 90.000,E1 313.218} C_DIS
LIN {X -0.079,Y -599.435,Z 1080.534,A 0.000,B 0.000,C 90.000,E1 312.162} C_DIS
LIN {X 0.348,Y -598.070,Z 1080.528,A 0.000,B 0.000,C 90.000,E1 311.067} C_DIS
LIN {X -0.254,Y -596.398,Z 1080.521,A 0.000,B 0.000,C 90.000,E1 309.806} C_DIS
LIN {X -0.267,Y -594.859,Z 1080.515,A 0.000,B 0.000,C 90.000,E1 308.749} C_DIS
LIN {X 0.155,Y -593.218,Z 1080.509,A 0.000,B 0.000,C 90.000,E1 307.649} C_DIS
LIN {X -0.074,Y -590.820,Z 1080.502,A 0.000,B 0.000,C 90.000,E1 306.343} C_DIS
LIN {X 0.065,Y -588.613,Z 1080.496,A 0.000,B 0.000,C 90.000,E1 305.264} C_DIS
LIN {X 0.040,Y -585.884,Z 1080.490,A 0.000,B 0.000,C 90.000,E1 304.199} C_DIS
LIN {X 0.271,Y -583.392,Z 1080.486,A 0.000,B 0.000,C 90.000,E1 303.372} C_DIS
LIN {X -0.358,Y -582.498,Z 1080.484,A 0.000,B 0.000,C 90.000,E1 303.166} C_DIS
LIN {X -0.016,Y -580.456,Z 1080.481,A 0.000,B 0.000,C 90.000,E1 302.594} C_DIS
LIN {X -0.084,Y -577.181,Z 1080.477,A 0.000,B 0.000,C 90.000,E1 301.926} C_DIS
LIN {X -0.178,Y -573.546,Z 1080.474,A 0.000,B 0.000,C 90.000,E1 301.258} C_DIS
LIN {X 0.275,Y -570.269,Z 1080.471,A 0.000,B 0.000,C 90.000,E1 300.669} C_DIS
LIN {X 0.210,Y -566.267,Z 1080.468,A 0.000,B 0.000,C 90.000,E1 300.129} C_DIS
LIN {X -0.068,Y -562.677,Z 1080.465,A 0.000,B 0.000,C 90.000,E1 299.745} C_DIS
LIN {X 0.087,Y -560.011,Z 1080.464,A 0.000,B 0.000,C 90.000,E1 299.461} C_DIS
LIN {X 0.058,Y -558.233,Z 1080.463,A 0.000,B 0.000,C 90.000,E1 299.333} C_DIS
LIN {X -0.083,Y -554.746,Z 1080.462,A 0.000,B 0.000,C 90.000,E1 299.127} C_DIS
LIN {X 0.199,Y -549.249,Z 1080.460,A 0.000,B 0.000,C 90.000,E1 298.693} C_DIS
LIN {X 0.015,Y -546.993,Z 1080.458,A 0.000,B 0.000,C 90.000,E1 298.487} C_DIS
LIN {X -0.150,Y -545.450,Z 1080.457,A 0.000,B 0.000,C 90.000,E1 298.281} C_DIS
LIN {X 0.097,Y -543.615,Z 1080.455,A 0.000,B 0.000,C 90.000,E1 297.897} C_DIS
LIN {X -0.027,Y -543.296,Z 1080.454,A 0.000,B 0.000,C 90.000,E1 297.769} C_DIS
LIN {X 0.200,Y -542.388,Z 1080.453,A 0.000,B 0.000,C 90.000,E1 297.462} C_DIS
LIN {X 0.072,Y -542.088,Z 1080.452,A 0.000,B 0.000,C 90.000,E1 297.334} C_DIS
LIN {X 0.157,Y -541.175,Z 1080.448,A 0.000,B 0.000,C 90.000,E1 296.616} C_DIS
LIN {X -0.288,Y -541.047,Z 1080.446,A 0.000,B 0.000,C 90.000,E1 296.232} C_DIS
LIN {X -0.244,Y -540.877,Z 1080.430,A 0.000,B 0.000,C 90.000,E1 293.387} C_DIS
LIN {X -0.061,Y -541.269,Z 1080.420,A 0.000,B 0.000,C 90.000,E1 291.663} C_DIS
LIN {X -0.099,Y -541.692,Z 1080.412,A 0.000,B 0.000,C 90.000,E1 290.248} C_DIS
LIN {X 0.140,Y -541.849,Z 1080.406,A 0.000,B 0.000,C 90.000,E1 289.087} C_DIS
LIN {X 0.206,Y -541.860,Z 1080.400,A 0.000,B 0.000,C 90.000,E1 287.946} C_DIS
LIN {X -0.022,Y -541.762,Z 1080.392,A 0.000,B 0.000,C 90.000,E1 286.551} C_DIS
LIN {X -0.043,Y -541.395,Z 1080.384,A 0.000,B 0.000,C 90.000,E1 285.134} C_DIS
LIN {X 0.071,Y -540.897,Z 1080.376,A 0.000,B 0.000,C 90.000,E1 283.703} C_DIS
LIN {X -0.085,Y -540.288,Z 1080.368,A 0.000,B 0.000,C 90.000,E1 282.299} C_DIS
LIN {X -0.246,Y -539.555,Z 1080.360,A 0.000,B 0.000,C 90.000,E1 280.894} C_DIS
LIN {X 0.213,Y -538.392,Z 1080.348,A 0.000,B 0.000,C 90.000,E1 278.568} C_DIS
LIN {X -0.111,Y -537.339,Z 1080.337,A 0.000,B 0.000,C 90.000,E1 276.606} C_DIS
LIN {X 0.030,Y -536.443,Z 1080.327,A 0.000,B 0.000,C 90.000,E1 274.878} C_DIS
LIN {X 0.107,Y -535.685,Z 1080.319,A 0.000,B 0.000,C 90.000,E1 273.440} C_DIS
LIN {X 0.155,Y -534.708,Z 1080.308,A 0.000,B 0.000,C 90.000,E1 271.432} C_DIS
LIN {X 0.152,Y -534.119,Z 1080.302,A 0.000,B 0.000,C 90.000,E1 270.286} C_DIS
LIN {X 0.138,Y -533.349,Z 1080.294,A 0.000,B 0.000,C 90.000,E1 268.854} C_DIS
LIN {X 0.110,Y -532.337,Z 1080.284,A 0.000,B 0.000,C 90.000,E1 267.135} C_DIS
LIN {X 0.106,Y -531.499,Z 1080.276,A 0.000,B 0.000,C 90.000,E1 265.698} C_DIS
LIN {X 0.089,Y -530.418,Z 1080.268,A 0.000,B 0.000,C 90.000,E1 264.261} C_DIS
LIN {X 0.104,Y -529.127,Z 1080.260,A 0.000,B 0.000,C 90.000,E1 262.818} C_DIS
LIN {X 0.115,Y -527.303,Z 1080.251,A 0.000,B 0.000,C 90.000,E1 261.084} C_DIS
LIN {X 0.142,Y -525.784,Z 1080.243,A 0.000,B 0.000,C 90.000,E1 259.634} C_DIS
LIN {X -0.265,Y -523.930,Z 1080.233,A 0.000,B 0.000,C 90.000,E1 257.937} C_DIS
LIN {X -0.083,Y -522.217,Z 1080.223,A 0.000,B 0.000,C 90.000,E1 256.172} C_DIS
LIN {X 0.180,Y -520.169,Z 1080.212,A 0.000,B 0.000,C 90.000,E1 254.102} C_DIS
LIN {X 0.045,Y -518.288,Z 1080.202,A 0.000,B 0.000,C 90.000,E1 252.362} C_DIS
LIN {X -0.232,Y -517.084,Z 1080.196,A 0.000,B 0.000,C 90.000,E1 251.221} C_DIS
LIN {X -0.229,Y -515.451,Z 1080.187,A 0.000,B 0.000,C 90.000,E1 249.752} C_DIS
LIN {X -0.128,Y -513.246,Z 1080.178,A 0.000,B 0.000,C 90.000,E1 247.975} C_DIS
LIN {X 0.108,Y -510.753,Z 1080.168,A 0.000,B 0.000,C 90.000,E1 246.177} C_DIS
LIN {X -0.034,Y -509.430,Z 1080.163,A 0.000,B 0.000,C 90.000,E1 245.305} C_DIS
LIN {X -0.022,Y -507.119,Z 1080.155,A 0.000,B 0.000,C 90.000,E1 243.819} C_DIS
LIN {X 0.100,Y -505.153,Z 1080.148,A 0.000,B 0.000,C 90.000,E1 242.615} C_DIS
LIN {X -0.026,Y -503.150,Z 1080.141,A 0.000,B 0.000,C 90.000,E1 241.435} C_DIS
LIN {X 0.029,Y -499.530,Z 1080.130,A 0.000,B 0.000,C 90.000,E1 239.331} C_DIS
LIN {X -0.049,Y -496.246,Z 1080.120,A 0.000,B 0.000,C 90.000,E1 237.533} C_DIS
LIN {X 0.063,Y -493.394,Z 1080.111,A 0.000,B 0.000,C 90.000,E1 236.008} C_DIS
LIN {X 0.125,Y -490.447,Z 1080.103,A 0.000,B 0.000,C 90.000,E1 234.482} C_DIS
LIN {X -0.144,Y -486.741,Z 1080.093,A 0.000,B 0.000,C 90.000,E1 232.683} C_DIS
LIN {X 0.185,Y -482.811,Z 1080.082,A 0.000,B 0.000,C 90.000,E1 230.803} C_DIS
LIN {X -0.017,Y -478.850,Z 1080.072,A 0.000,B 0.000,C 90.000,E1 228.976} C_DIS
LIN {X 0.150,Y -474.427,Z 1080.060,A 0.000,B 0.000,C 90.000,E1 226.782} C_DIS
LIN {X 0.060,Y -470.958,Z 1080.050,A 0.000,B 0.000,C 90.000,E1 224.919} C_DIS
LIN {X -0.108,Y -467.456,Z 1080.039,A 0.000,B 0.000,C 90.000,E1 223.056} C_DIS
LIN {X 0.131,Y -465.675,Z 1080.034,A 0.000,B 0.000,C 90.000,E1 222.081} C_DIS
LIN {X -0.045,Y -461.366,Z 1080.022,A 0.000,B 0.000,C 90.000,E1 219.886} C_DIS
LIN {X -0.104,Y -458.331,Z 1080.013,A 0.000,B 0.000,C 90.000,E1 218.302} C_DIS
LIN {X -0.063,Y -454.579,Z 1080.002,A 0.000,B 0.000,C 90.000,E1 216.377} C_DIS
LIN {X 0.175,Y -451.418,Z 1079.993,A 0.000,B 0.000,C 90.000,E1 214.739} C_DIS
LIN {X 0.063,Y -446.497,Z 1079.979,A 0.000,B 0.000,C 90.000,E1 212.163} C_DIS
LIN {X 0.017,Y -443.545,Z 1079.970,A 0.000,B 0.000,C 90.000,E1 210.541} C_DIS
LIN {X 0.156,Y -439.397,Z 1079.957,A 0.000,B 0.000,C 90.000,E1 208.231} C_DIS
LIN {X -0.237,Y -435.455,Z 1079.944,A 0.000,B 0.000,C 90.000,E1 205.976} C_DIS
LIN {X 0.043,Y -433.009,Z 1079.935,A 0.000,B 0.000,C 90.000,E1 204.283} C_DIS
LIN {X -0.123,Y -429.438,Z 1079.920,A 0.000,B 0.000,C 90.000,E1 201.642} C_DIS
LIN {X 0.112,Y -428.066,Z 1079.911,A 0.000,B 0.000,C 90.000,E1 199.939} C_DIS
LIN {X 0.120,Y -427.922,Z 1079.907,A 0.000,B 0.000,C 90.000,E1 199.268} C_DIS
LIN {X 0.125,Y -428.050,Z 1079.903,A 0.000,B 0.000,C 90.000,E1 198.598} C_DIS
LIN {X -0.004,Y -428.560,Z 1079.900,A 0.000,B 0.000,C 90.000,E1 197.946} C_DIS
LIN {X 0.002,Y -429.474,Z 1079.896,A 0.000,B 0.000,C 90.000,E1 197.275} C_DIS
LIN {X -0.114,Y -430.876,Z 1079.892,A 0.000,B 0.000,C 90.000,E1 196.622} C_DIS
LIN {X 0.100,Y -431.729,Z 1079.891,A 0.000,B 0.000,C 90.000,E1 196.260} C_DIS
LIN {X 0.115,Y -434.400,Z 1079.886,A 0.000,B 0.000,C 90.000,E1 195.426} C_DIS
LIN {X -0.177,Y -442.118,Z 1079.876,A 0.000,B 0.000,C 90.000,E1 193.647} C_DIS
LIN {X -0.156,Y -449.140,Z 1079.868,A 0.000,B 0.000,C 90.000,E1 192.175} C_DIS
LIN {X -0.034,Y -460.912,Z 1079.855,A 0.000,B 0.000,C 90.000,E1 189.905} C_DIS
LIN {X 0.156,Y -468.747,Z 1079.847,A 0.000,B 0.000,C 90.000,E1 188.454} C_DIS
LIN {X -0.170,Y -475.676,Z 1079.840,A 0.000,B 0.000,C 90.000,E1 187.239} C_DIS
LIN {X 0.098,Y -479.879,Z 1079.836,A 0.000,B 0.000,C 90.000,E1 186.429} C_DIS
LIN {X 0.209,Y -485.512,Z 1079.830,A 0.000,B 0.000,C 90.000,E1 185.334} C_DIS
LIN {X -0.129,Y -491.133,Z 1079.824,A 0.000,B 0.000,C 90.000,E1 184.302} C_DIS
LIN {X -0.074,Y -495.808,Z 1079.819,A 0.000,B 0.000,C 90.000,E1 183.383} C_DIS
LIN {X 0.097,Y -502.795,Z 1079.811,A 0.000,B 0.000,C 90.000,E1 182.007} C_DIS
LIN {X 0.088,Y -510.370,Z 1079.803,A 0.000,B 0.000,C 90.000,E1 180.516} C_DIS
LIN {X -0.083,Y -518.727,Z 1079.794,A 0.000,B 0.000,C 90.000,E1 178.912} C_DIS
LIN {X -0.080,Y -526.897,Z 1079.785,A 0.000,B 0.000,C 90.000,E1 177.306} C_DIS
LIN {X -0.139,Y -534.259,Z 1079.777,A 0.000,B 0.000,C 90.000,E1 175.869} C_DIS
LIN {X -0.060,Y -541.573,Z 1079.769,A 0.000,B 0.000,C 90.000,E1 174.432} C_DIS
LIN {X -0.140,Y -548.048,Z 1079.762,A 0.000,B 0.000,C 90.000,E1 173.166} C_DIS
LIN {X 0.066,Y -555.851,Z 1079.753,A 0.000,B 0.000,C 90.000,E1 171.602} C_DIS
LIN {X 0.125,Y -562.763,Z 1079.746,A 0.000,B 0.000,C 90.000,E1 170.208} C_DIS
LIN {X -0.117,Y -568.775,Z 1079.739,A 0.000,B 0.000,C 90.000,E1 168.993} C_DIS
LIN {X -0.052,Y -574.527,Z 1079.732,A 0.000,B 0.000,C 90.000,E1 167.757} C_DIS
LIN {X -0.226,Y -581.275,Z 1079.724,A 0.000,B 0.000,C 90.000,E1 166.284} C_DIS
LIN {X 0.043,Y -586.573,Z 1079.717,A 0.000,B 0.000,C 90.000,E1 165.046} C_DIS
LIN {X 0.050,Y -590.903,Z 1079.711,A 0.000,B 0.000,C 90.000,E1 163.976} C_DIS
LIN {X -0.148,Y -594.039,Z 1079.707,A 0.000,B 0.000,C 90.000,E1 163.196} C_DIS
LIN {X -0.044,Y -598.004,Z 1079.701,A 0.000,B 0.000,C 90.000,E1 162.127} C_DIS
LIN {X -0.276,Y -601.780,Z 1079.695,A 0.000,B 0.000,C 90.000,E1 161.094} C_DIS
LIN {X 0.115,Y -605.287,Z 1079.689,A 0.000,B 0.000,C 90.000,E1 160.007} C_DIS
LIN {X -0.083,Y -609.404,Z 1079.682,A 0.000,B 0.000,C 90.000,E1 158.720} C_DIS
LIN {X 0.019,Y -613.276,Z 1079.675,A 0.000,B 0.000,C 90.000,E1 157.411} C_DIS
LIN {X 0.193,Y -616.983,Z 1079.667,A 0.000,B 0.000,C 90.000,E1 156.102} C_DIS
LIN {X -0.149,Y -621.679,Z 1079.657,A 0.000,B 0.000,C 90.000,E1 154.332} C_DIS
LIN {X -0.141,Y -624.304,Z 1079.652,A 0.000,B 0.000,C 90.000,E1 153.307} C_DIS
LIN {X -0.069,Y -627.988,Z 1079.643,A 0.000,B 0.000,C 90.000,E1 151.769} C_DIS
LIN {X 0.317,Y -630.361,Z 1079.638,A 0.000,B 0.000,C 90.000,E1 150.717} C_DIS
LIN {X 0.252,Y -633.739,Z 1079.629,A 0.000,B 0.000,C 90.000,E1 149.203} C_DIS
LIN {X 0.070,Y -637.525,Z 1079.619,A 0.000,B 0.000,C 90.000,E1 147.454} C_DIS
LIN {X -0.215,Y -641.123,Z 1079.609,A 0.000,B 0.000,C 90.000,E1 145.722} C_DIS
LIN {X -0.420,Y -644.567,Z 1079.600,A 0.000,B 0.000,C 90.000,E1 143.989} C_DIS
LIN {X -0.272,Y -648.382,Z 1079.589,A 0.000,B 0.000,C 90.000,E1 141.984} C_DIS
LIN {X 0.036,Y -650.343,Z 1079.583,A 0.000,B 0.000,C 90.000,E1 140.964} C_DIS
LIN {X 0.253,Y -653.290,Z 1079.575,A 0.000,B 0.000,C 90.000,E1 139.461} C_DIS
LIN {X 0.042,Y -656.346,Z 1079.567,A 0.000,B 0.000,C 90.000,E1 138.000} C_DIS
LIN {X -0.185,Y -661.021,Z 1079.554,A 0.000,B 0.000,C 90.000,E1 135.810} C_DIS
LIN {X -0.271,Y -664.512,Z 1079.546,A 0.000,B 0.000,C 90.000,E1 134.352} C_DIS
LIN {X 0.199,Y -670.052,Z 1079.534,A 0.000,B 0.000,C 90.000,E1 132.123} C_DIS
LIN {X -0.130,Y -673.766,Z 1079.526,A 0.000,B 0.000,C 90.000,E1 130.701} C_DIS
LIN {X -0.382,Y -677.439,Z 1079.518,A 0.000,B 0.000,C 90.000,E1 129.277} C_DIS
LIN {X -0.016,Y -681.721,Z 1079.509,A 0.000,B 0.000,C 90.000,E1 127.569} C_DIS
LIN {X -0.039,Y -684.859,Z 1079.502,A 0.000,B 0.000,C 90.000,E1 126.377} C_DIS
LIN {X -0.214,Y -686.668,Z 1079.498,A 0.000,B 0.000,C 90.000,E1 125.678} C_DIS
LIN {X -0.121,Y -690.110,Z 1079.490,A 0.000,B 0.000,C 90.000,E1 124.246} C_DIS
LIN {X -0.170,Y -693.582,Z 1079.482,A 0.000,B 0.000,C 90.000,E1 122.832} C_DIS
LIN {X 0.226,Y -696.979,Z 1079.474,A 0.000,B 0.000,C 90.000,E1 121.386} C_DIS
LIN {X 0.038,Y -699.020,Z 1079.469,A 0.000,B 0.000,C 90.000,E1 120.463} C_DIS
LIN {X -0.045,Y -699.957,Z 1079.467,A 0.000,B 0.000,C 90.000,E1 120.001} C_DIS
LIN {X 0.148,Y -701.018,Z 1079.463,A 0.000,B 0.000,C 90.000,E1 119.283} C_DIS
LIN {X 0.013,Y -702.049,Z 1079.458,A 0.000,B 0.000,C 90.000,E1 118.359} C_DIS
LIN {X -0.222,Y -703.634,Z 1079.448,A 0.000,B 0.000,C 90.000,E1 116.744} C_DIS
LIN {X 0.263,Y -704.710,Z 1079.442,A 0.000,B 0.000,C 90.000,E1 115.540} C_DIS
LIN {X 0.201,Y -705.023,Z 1079.439,A 0.000,B 0.000,C 90.000,E1 115.079} C_DIS
LIN {X -0.162,Y -705.108,Z 1079.437,A 0.000,B 0.000,C 90.000,E1 114.643} C_DIS
LIN {X 0.123,Y -704.650,Z 1079.434,A 0.000,B 0.000,C 90.000,E1 114.155} C_DIS
LIN {X -0.234,Y -704.269,Z 1079.433,A 0.000,B 0.000,C 90.000,E1 113.951} C_DIS
LIN {X 0.049,Y -702.655,Z 1079.430,A 0.000,B 0.000,C 90.000,E1 113.462} C_DIS
LIN {X 0.328,Y -701.437,Z 1079.429,A 0.000,B 0.000,C 90.000,E1 113.206} C_DIS
LIN {X -0.049,Y -697.815,Z 1079.427,A 0.000,B 0.000,C 90.000,E1 112.770} C_DIS
LIN {X 0.080,Y -696.547,Z 1079.426,A 0.000,B 0.000,C 90.000,E1 112.642} C_DIS
LIN {X 0.209,Y -694.536,Z 1079.425,A 0.000,B 0.000,C 90.000,E1 112.514} C_DIS
LIN {X 0.104,Y -687.322,Z 1079.423,A 0.000,B 0.000,C 90.000,E1 112.206} C_DIS
LIN {X -0.117,Y -685.174,Z 1079.423,A 0.000,B 0.000,C 90.000,E1 112.153} C_DIS
LIN {X -0.074,Y -676.347,Z 1079.422,A 0.000,B 0.000,C 90.000,E1 112.025} C_DIS
LIN {X -0.138,Y -669.373,Z 1079.422,A 0.000,B 0.000,C 90.000,E1 112.025} C_DIS
LIN {X -0.175,Y -605.896,Z 1079.422,A 0.000,B 0.000,C 90.000,E1 112.025} C_DIS
LIN {X -0.156,Y -601.908,Z 1079.421,A 0.000,B 0.000,C 90.000,E1 111.844} C_DIS
LIN {X 0.107,Y -596.543,Z 1079.419,A 0.000,B 0.000,C 90.000,E1 111.482} C_DIS
LIN {X 0.090,Y -588.722,Z 1079.416,A 0.000,B 0.000,C 90.000,E1 110.865} C_DIS
LIN {X -0.050,Y -579.106,Z 1079.411,A 0.000,B 0.000,C 90.000,E1 110.066} C_DIS
LIN {X 0.166,Y -574.931,Z 1079.410,A 0.000,B 0.000,C 90.000,E1 109.704} C_DIS
LIN {X 0.000,Y -568.852,Z 1079.407,A 0.000,B 0.000,C 90.000,E1 109.268} C_DIS
LIN {X -0.236,Y -560.507,Z 1079.404,A 0.000,B 0.000,C 90.000,E1 108.779} C_DIS
LIN {X -0.223,Y -554.135,Z 1079.402,A 0.000,B 0.000,C 90.000,E1 108.417} C_DIS
LIN {X -0.174,Y -549.718,Z 1079.401,A 0.000,B 0.000,C 90.000,E1 108.109} C_DIS
LIN {X -0.138,Y -548.731,Z 1079.400,A 0.000,B 0.000,C 90.000,E1 108.000} C_DIS
LIN {X -0.100,Y -547.770,Z 1079.399,A 0.000,B 0.000,C 90.000,E1 107.873} C_DIS
LIN {X -0.142,Y -547.755,Z 1079.399,A 0.000,B 0.000,C 90.000,E1 107.873} C_DIS
LIN {X 0.156,Y -547.402,Z 1079.398,A 0.000,B 0.000,C 90.000,E1 107.583} C_DIS
LIN {X -0.220,Y -548.683,Z 1079.385,A 0.000,B 0.000,C 90.000,E1 105.371} C_DIS
LIN {X 0.246,Y -550.153,Z 1079.374,A 0.000,B 0.000,C 90.000,E1 103.355} C_DIS
LIN {X -0.272,Y -551.310,Z 1079.367,A 0.000,B 0.000,C 90.000,E1 102.007} C_DIS
LIN {X 0.008,Y -553.192,Z 1079.356,A 0.000,B 0.000,C 90.000,E1 100.018} C_DIS
LIN {X 0.147,Y -555.365,Z 1079.345,A 0.000,B 0.000,C 90.000,E1 98.049} C_DIS
LIN {X 0.210,Y -557.212,Z 1079.336,A 0.000,B 0.000,C 90.000,E1 96.372} C_DIS
LIN {X 0.117,Y -558.650,Z 1079.328,A 0.000,B 0.000,C 90.000,E1 94.992} C_DIS
LIN {X -0.034,Y -559.549,Z 1079.322,A 0.000,B 0.000,C 90.000,E1 93.898} C_DIS
LIN {X -0.126,Y -560.357,Z 1079.314,A 0.000,B 0.000,C 90.000,E1 92.522} C_DIS
LIN {X -0.201,Y -561.113,Z 1079.306,A 0.000,B 0.000,C 90.000,E1 91.146} C_DIS
LIN {X -0.275,Y -561.673,Z 1079.299,A 0.000,B 0.000,C 90.000,E1 89.771} C_DIS
LIN {X -0.227,Y -562.337,Z 1079.289,A 0.000,B 0.000,C 90.000,E1 88.108} C_DIS
LIN {X -0.261,Y -562.871,Z 1079.282,A 0.000,B 0.000,C 90.000,E1 86.731} C_DIS
LIN {X -0.295,Y -563.427,Z 1079.274,A 0.000,B 0.000,C 90.000,E1 85.355} C_DIS
LIN {X -0.137,Y -563.963,Z 1079.265,A 0.000,B 0.000,C 90.000,E1 83.685} C_DIS
LIN {X -0.056,Y -564.389,Z 1079.257,A 0.000,B 0.000,C 90.000,E1 82.299} C_DIS
LIN {X -0.202,Y -565.032,Z 1079.247,A 0.000,B 0.000,C 90.000,E1 80.387} C_DIS
LIN {X -0.240,Y -565.867,Z 1079.236,A 0.000,B 0.000,C 90.000,E1 78.465} C_DIS
LIN {X -0.226,Y -567.145,Z 1079.222,A 0.000,B 0.000,C 90.000,E1 75.992} C_DIS
LIN {X -0.199,Y -568.545,Z 1079.210,A 0.000,B 0.000,C 90.000,E1 73.795} C_DIS
LIN {X -0.111,Y -569.656,Z 1079.202,A 0.000,B 0.000,C 90.000,E1 72.417} C_DIS
LIN {X -0.202,Y -570.991,Z 1079.193,A 0.000,B 0.000,C 90.000,E1 70.786} C_DIS
LIN {X -0.073,Y -572.368,Z 1079.184,A 0.000,B 0.000,C 90.000,E1 69.135} C_DIS
LIN {X -0.089,Y -573.964,Z 1079.173,A 0.000,B 0.000,C 90.000,E1 67.230} C_DIS
LIN {X -0.228,Y -575.218,Z 1079.164,A 0.000,B 0.000,C 90.000,E1 65.613} C_DIS
LIN {X -0.327,Y -575.942,Z 1079.158,A 0.000,B 0.000,C 90.000,E1 64.537} C_DIS
LIN {X -0.159,Y -576.589,Z 1079.152,A 0.000,B 0.000,C 90.000,E1 63.435} C_DIS
LIN {X -0.119,Y -577.414,Z 1079.145,A 0.000,B 0.000,C 90.000,E1 62.076} C_DIS
LIN {X -0.216,Y -578.396,Z 1079.136,A 0.000,B 0.000,C 90.000,E1 60.461} C_DIS
LIN {X 0.126,Y -579.039,Z 1079.128,A 0.000,B 0.000,C 90.000,E1 59.076} C_DIS
LIN {X 0.127,Y -579.610,Z 1079.122,A 0.000,B 0.000,C 90.000,E1 57.995} C_DIS
LIN {X 0.299,Y -580.214,Z 1079.115,A 0.000,B 0.000,C 90.000,E1 56.628} C_DIS
LIN {X 0.005,Y -581.086,Z 1079.104,A 0.000,B 0.000,C 90.000,E1 54.769} C_DIS
LIN {X 0.225,Y -581.497,Z 1079.095,A 0.000,B 0.000,C 90.000,E1 53.130} C_DIS
LIN {X 0.103,Y -581.646,Z 1079.089,A 0.000,B 0.000,C 90.000,E1 52.065} C_DIS
LIN {X -0.008,Y -581.665,Z 1079.086,A 0.000,B 0.000,C 90.000,E1 51.537} C_DIS
LIN {X -0.116,Y -581.675,Z 1079.083,A 0.000,B 0.000,C 90.000,E1 51.009} C_DIS
LIN {X 0.015,Y -581.216,Z 1079.074,A 0.000,B 0.000,C 90.000,E1 49.380} C_DIS
LIN {X -0.204,Y -580.830,Z 1079.068,A 0.000,B 0.000,C 90.000,E1 48.324} C_DIS
LIN {X -0.159,Y -580.031,Z 1079.059,A 0.000,B 0.000,C 90.000,E1 46.701} C_DIS
LIN {X -0.014,Y -579.313,Z 1079.053,A 0.000,B 0.000,C 90.000,E1 45.607} C_DIS
LIN {X 0.117,Y -578.377,Z 1079.047,A 0.000,B 0.000,C 90.000,E1 44.514} C_DIS
LIN {X -0.174,Y -577.192,Z 1079.041,A 0.000,B 0.000,C 90.000,E1 43.461} C_DIS
LIN {X 0.076,Y -575.391,Z 1079.034,A 0.000,B 0.000,C 90.000,E1 42.081} C_DIS
LIN {X 0.019,Y -574.183,Z 1079.029,A 0.000,B 0.000,C 90.000,E1 41.272} C_DIS
LIN {X 0.136,Y -572.176,Z 1079.023,A 0.000,B 0.000,C 90.000,E1 40.172} C_DIS
LIN {X -0.208,Y -569.943,Z 1079.017,A 0.000,B 0.000,C 90.000,E1 39.116} C_DIS
LIN {X 0.178,Y -568.015,Z 1079.013,A 0.000,B 0.000,C 90.000,E1 38.257} C_DIS
LIN {X -0.022,Y -566.621,Z 1079.010,A 0.000,B 0.000,C 90.000,E1 37.729} C_DIS
LIN {X 0.329,Y -564.189,Z 1079.005,A 0.000,B 0.000,C 90.000,E1 36.870} C_DIS
LIN {X -0.132,Y -561.542,Z 1079.000,A 0.000,B 0.000,C 90.000,E1 36.091} C_DIS
LIN {X 0.067,Y -559.511,Z 1078.997,A 0.000,B 0.000,C 90.000,E1 35.518} C_DIS
LIN {X -0.071,Y -557.268,Z 1078.994,A 0.000,B 0.000,C 90.000,E1 34.978} C_DIS
LIN {X 0.052,Y -553.093,Z 1078.989,A 0.000,B 0.000,C 90.000,E1 33.992} C_DIS
LIN {X 0.055,Y -549.841,Z 1078.985,A 0.000,B 0.000,C 90.000,E1 33.293} C_DIS
LIN {X -0.234,Y -544.922,Z 1078.980,A 0.000,B 0.000,C 90.000,E1 32.339} C_DIS
LIN {X -0.120,Y -539.530,Z 1078.974,A 0.000,B 0.000,C 90.000,E1 31.337} C_DIS
LIN {X 0.066,Y -534.610,Z 1078.969,A 0.000,B 0.000,C 90.000,E1 30.463} C_DIS
LIN {X 0.222,Y -531.069,Z 1078.966,A 0.000,B 0.000,C 90.000,E1 29.873} C_DIS
LIN {X -0.261,Y -526.118,Z 1078.962,A 0.000,B 0.000,C 90.000,E1 29.205} C_DIS
LIN {X -0.166,Y -521.913,Z 1078.959,A 0.000,B 0.000,C 90.000,E1 28.615} C_DIS
LIN {X 0.189,Y -516.313,Z 1078.955,A 0.000,B 0.000,C 90.000,E1 27.847} C_DIS
LIN {X 0.085,Y -510.324,Z 1078.951,A 0.000,B 0.000,C 90.000,E1 27.129} C_DIS
LIN {X -0.052,Y -505.172,Z 1078.948,A 0.000,B 0.000,C 90.000,E1 26.565} C_DIS
LIN {X 0.143,Y -495.686,Z 1078.942,A 0.000,B 0.000,C 90.000,E1 25.540} C_DIS
LIN {X -0.250,Y -484.432,Z 1078.936,A 0.000,B 0.000,C 90.000,E1 24.463} C_DIS
LIN {X 0.167,Y -474.319,Z 1078.931,A 0.000,B 0.000,C 90.000,E1 23.462} C_DIS
LIN {X -0.068,Y -464.039,Z 1078.926,A 0.000,B 0.000,C 90.000,E1 22.589} C_DIS
LIN {X -0.035,Y -450.449,Z 1078.919,A 0.000,B 0.000,C 90.000,E1 21.408} C_DIS
LIN {X 0.107,Y -429.970,Z 1078.908,A 0.000,B 0.000,C 90.000,E1 19.504} C_DIS
LIN {X 0.074,Y -417.137,Z 1078.901,A 0.000,B 0.000,C 90.000,E1 18.181} C_DIS
LIN {X 0.201,Y -406.371,Z 1078.894,A 0.000,B 0.000,C 90.000,E1 16.913} C_DIS
LIN {X -0.095,Y -400.032,Z 1078.890,A 0.000,B 0.000,C 90.000,E1 16.134} C_DIS
LIN {X 0.138,Y -396.042,Z 1078.886,A 0.000,B 0.000,C 90.000,E1 15.481} C_DIS
LIN {X 0.090,Y -393.370,Z 1078.883,A 0.000,B 0.000,C 90.000,E1 14.898} C_DIS
LIN {X 0.143,Y -392.547,Z 1078.881,A 0.000,B 0.000,C 90.000,E1 14.537} C_DIS
LIN {X 0.168,Y -392.275,Z 1078.880,A 0.000,B 0.000,C 90.000,E1 14.356} C_DIS
LIN {X 0.053,Y -391.874,Z 1078.877,A 0.000,B 0.000,C 90.000,E1 13.828} C_DIS
LIN {X 0.042,Y -392.304,Z 1078.873,A 0.000,B 0.000,C 90.000,E1 13.119} C_DIS
LIN {X -0.098,Y -394.610,Z 1078.863,A 0.000,B 0.000,C 90.000,E1 11.366} C_DIS
LIN {X 0.101,Y -400.957,Z 1078.844,A 0.000,B 0.000,C 90.000,E1 7.814} C_DIS
LIN {X -0.041,Y -405.549,Z 1078.832,A 0.000,B 0.000,C 90.000,E1 5.739} C_DIS
LIN {X -0.076,Y -406.991,Z 1078.828,A 0.000,B 0.000,C 90.000,E1 5.049} C_DIS
LIN {X -0.099,Y -408.968,Z 1078.824,A 0.000,B 0.000,C 90.000,E1 4.359} C_DIS
LIN {X -0.092,Y -410.394,Z 1078.822,A 0.000,B 0.000,C 90.000,E1 4.012} C_DIS
LIN {X 0.097,Y -412.423,Z 1078.820,A 0.000,B 0.000,C 90.000,E1 3.555} C_DIS
LIN {X 0.004,Y -417.401,Z 1078.817,A 0.000,B 0.000,C 90.000,E1 2.980} C_DIS
LIN {X -0.033,Y -421.158,Z 1078.815,A 0.000,B 0.000,C 90.000,E1 2.694} C_DIS
LIN {X 0.118,Y -430.505,Z 1078.812,A 0.000,B 0.000,C 90.000,E1 2.064} C_DIS
LIN {X 0.204,Y -456.939,Z 1078.802,A 0.000,B 0.000,C 90.000,E1 0.344} C_DIS
LIN {X 0.162,Y -472.693,Z 1078.797,A 0.000,B 0.000,C 90.000,E1 359.370} C_DIS
LIN {X -0.041,Y -484.170,Z 1078.793,A 0.000,B 0.000,C 90.000,E1 358.682} C_DIS
LIN {X 0.117,Y -495.310,Z 1078.789,A 0.000,B 0.000,C 90.000,E1 357.936} C_DIS
LIN {X -0.070,Y -503.121,Z 1078.786,A 0.000,B 0.000,C 90.000,E1 357.421} C_DIS
LIN {X 0.034,Y -512.254,Z 1078.782,A 0.000,B 0.000,C 90.000,E1 356.731} C_DIS
LIN {X 0.007,Y -516.770,Z 1078.780,A 0.000,B 0.000,C 90.000,E1 356.388} C_DIS
LIN {X -0.209,Y -523.861,Z 1078.777,A 0.000,B 0.000,C 90.000,E1 355.812} C_DIS
LIN {X -0.208,Y -530.522,Z 1078.773,A 0.000,B 0.000,C 90.000,E1 355.179} C_DIS
LIN {X 0.111,Y -534.171,Z 1078.771,A 0.000,B 0.000,C 90.000,E1 354.780} C_DIS
LIN {X -0.162,Y -539.229,Z 1078.768,A 0.000,B 0.000,C 90.000,E1 354.261} C_DIS
LIN {X 0.213,Y -545.167,Z 1078.764,A 0.000,B 0.000,C 90.000,E1 353.514} C_DIS
LIN {X 0.033,Y -548.588,Z 1078.762,A 0.000,B 0.000,C 90.000,E1 353.109} C_DIS
LIN {X -0.025,Y -553.491,Z 1078.758,A 0.000,B 0.000,C 90.000,E1 352.413} C_DIS
LIN {X -0.113,Y -557.892,Z 1078.754,A 0.000,B 0.000,C 90.000,E1 351.724} C_DIS
LIN {X 0.161,Y -561.097,Z 1078.751,A 0.000,B 0.000,C 90.000,E1 351.141} C_DIS
LIN {X 0.048,Y -565.353,Z 1078.746,A 0.000,B 0.000,C 90.000,E1 350.330} C_DIS
LIN {X 0.141,Y -568.645,Z 1078.743,A 0.000,B 0.000,C 90.000,E1 349.634} C_DIS
LIN {X 0.131,Y -572.191,Z 1078.738,A 0.000,B 0.000,C 90.000,E1 348.814} C_DIS
LIN {X 0.159,Y -575.581,Z 1078.733,A 0.000,B 0.000,C 90.000,E1 347.993} C_DIS
LIN {X 0.222,Y -578.752,Z 1078.729,A 0.000,B 0.000,C 90.000,E1 347.173} C_DIS
LIN {X -0.023,Y -582.750,Z 1078.723,A 0.000,B 0.000,C 90.000,E1 346.117} C_DIS
LIN {X 0.168,Y -587.453,Z 1078.715,A 0.000,B 0.000,C 90.000,E1 344.755} C_DIS
LIN {X 0.183,Y -590.957,Z 1078.709,A 0.000,B 0.000,C 90.000,E1 343.685} C_DIS
LIN {X 0.113,Y -595.214,Z 1078.702,A 0.000,B 0.000,C 90.000,E1 342.362} C_DIS
LIN {X -0.153,Y -598.482,Z 1078.696,A 0.000,B 0.000,C 90.000,E1 341.329} C_DIS
LIN {X 0.193,Y -601.296,Z 1078.690,A 0.000,B 0.000,C 90.000,E1 340.242} C_DIS
LIN {X 0.008,Y -604.055,Z 1078.685,A 0.000,B 0.000,C 90.000,E1 339.209} C_DIS
LIN {X 0.140,Y -605.883,Z 1078.680,A 0.000,B 0.000,C 90.000,E1 338.411} C_DIS
LIN {X 0.231,Y -608.060,Z 1078.674,A 0.000,B 0.000,C 90.000,E1 337.358} C_DIS
LIN {X -0.161,Y -609.578,Z 1078.670,A 0.000,B 0.000,C 90.000,E1 336.613} C_DIS
LIN {X 0.225,Y -611.281,Z 1078.664,A 0.000,B 0.000,C 90.000,E1 335.537} C_DIS
LIN {X -0.207,Y -613.121,Z 1078.657,A 0.000,B 0.000,C 90.000,E1 334.280} C_DIS
LIN {X 0.201,Y -614.684,Z 1078.650,A 0.000,B 0.000,C 90.000,E1 332.948} C_DIS
LIN {X 0.124,Y -615.446,Z 1078.646,A 0.000,B 0.000,C 90.000,E1 332.180} C_DIS
LIN {X -0.216,Y -616.346,Z 1078.640,A 0.000,B 0.000,C 90.000,E1 331.179} C_DIS
LIN {X 0.024,Y -616.782,Z 1078.635,A 0.000,B 0.000,C 90.000,E1 330.383} C_DIS
LIN {X 0.250,Y -617.094,Z 1078.630,A 0.000,B 0.000,C 90.000,E1 329.331} C_DIS
LIN {X -0.030,Y -617.133,Z 1078.625,A 0.000,B 0.000,C 90.000,E1 328.584} C_DIS
LIN {X -0.034,Y -616.702,Z 1078.618,A 0.000,B 0.000,C 90.000,E1 327.296} C_DIS
LIN {X 0.201,Y -616.189,Z 1078.614,A 0.000,B 0.000,C 90.000,E1 326.501} C_DIS
LIN {X 0.004,Y -615.003,Z 1078.607,A 0.000,B 0.000,C 90.000,E1 325.229} C_DIS
LIN {X 0.325,Y -612.763,Z 1078.595,A 0.000,B 0.000,C 90.000,E1 323.130} C_DIS
LIN {X -0.129,Y -611.202,Z 1078.587,A 0.000,B 0.000,C 90.000,E1 321.618} C_DIS
LIN {X 0.040,Y -609.624,Z 1078.577,A 0.000,B 0.000,C 90.000,E1 319.784} C_DIS
LIN {X -0.171,Y -608.378,Z 1078.568,A 0.000,B 0.000,C 90.000,E1 318.243} C_DIS
LIN {X -0.282,Y -607.735,Z 1078.564,A 0.000,B 0.000,C 90.000,E1 317.472} C_DIS
LIN {X 0.014,Y -606.878,Z 1078.559,A 0.000,B 0.000,C 90.000,E1 316.662} C_DIS
LIN {X -0.066,Y -605.422,Z 1078.552,A 0.000,B 0.000,C 90.000,E1 315.364} C_DIS
LIN {X 0.167,Y -605.022,Z 1078.551,A 0.000,B 0.000,C 90.000,E1 315.081} C_DIS
LIN {X -0.220,Y -604.655,Z 1078.548,A 0.000,B 0.000,C 90.000,E1 314.595} C_DIS
LIN {X 0.007,Y -604.164,Z 1078.546,A 0.000,B 0.000,C 90.000,E1 314.312} C_DIS
LIN {X 0.087,Y -603.798,Z 1078.543,A 0.000,B 0.000,C 90.000,E1 313.785} C_DIS
LIN {X 0.169,Y -602.160,Z 1078.535,A 0.000,B 0.000,C 90.000,E1 312.204} C_DIS
LIN {X 0.233,Y -600.972,Z 1078.529,A 0.000,B 0.000,C 90.000,E1 311.148} C_DIS
LIN {X -0.290,Y -598.348,Z 1078.516,A 0.000,B 0.000,C 90.000,E1 308.830} C_DIS
LIN {X -0.186,Y -596.238,Z 1078.507,A 0.000,B 0.000,C 90.000,E1 307.237} C_DIS
LIN {X 0.125,Y -594.347,Z 1078.500,A 0.000,B 0.000,C 90.000,E1 305.884} C_DIS
LIN {X -0.257,Y -593.544,Z 1078.497,A 0.000,B 0.000,C 90.000,E1 305.391} C_DIS
LIN {X -0.008,Y -590.808,Z 1078.489,A 0.000,B 0.000,C 90.000,E1 304.040} C_DIS
LIN {X 0.149,Y -588.223,Z 1078.483,A 0.000,B 0.000,C 90.000,E1 302.959} C_DIS
LIN {X 0.090,Y -585.776,Z 1078.479,A 0.000,B 0.000,C 90.000,E1 302.163} C_DIS
LIN {X -0.353,Y -583.561,Z 1078.476,A 0.000,B 0.000,C 90.000,E1 301.671} C_DIS
LIN {X -0.248,Y -581.814,Z 1078.474,A 0.000,B 0.000,C 90.000,E1 301.258} C_DIS
LIN {X 0.199,Y -578.612,Z 1078.470,A 0.000,B 0.000,C 90.000,E1 300.541} C_DIS
LIN {X 0.195,Y -575.754,Z 1078.467,A 0.000,B 0.000,C 90.000,E1 300.001} C_DIS
LIN {X 0.167,Y -572.519,Z 1078.464,A 0.000,B 0.000,C 90.000,E1 299.461} C_DIS
LIN {X -0.081,Y -569.336,Z 1078.462,A 0.000,B 0.000,C 90.000,E1 299.077} C_DIS
LIN {X -0.336,Y -565.622,Z 1078.459,A 0.000,B 0.000,C 90.000,E1 298.693} C_DIS
LIN {X -0.108,Y -561.029,Z 1078.457,A 0.000,B 0.000,C 90.000,E1 298.281} C_DIS
LIN {X 0.091,Y -558.036,Z 1078.456,A 0.000,B 0.000,C 90.000,E1 298.025} C_DIS
LIN {X 0.195,Y -555.501,Z 1078.455,A 0.000,B 0.000,C 90.000,E1 297.897} C_DIS
LIN {X -0.073,Y -552.659,Z 1078.454,A 0.000,B 0.000,C 90.000,E1 297.769} C_DIS
LIN {X -0.030,Y -548.196,Z 1078.452,A 0.000,B 0.000,C 90.000,E1 297.385} C_DIS
LIN {X 0.037,Y -545.296,Z 1078.450,A 0.000,B 0.000,C 90.000,E1 297.001} C_DIS
LIN {X 0.018,Y -544.904,Z 1078.449,A 0.000,B 0.000,C 90.000,E1 296.873} C_DIS
LIN {X -0.229,Y -543.631,Z 1078.448,A 0.000,B 0.000,C 90.000,E1 296.616} C_DIS
LIN {X 0.006,Y -543.230,Z 1078.446,A 0.000,B 0.000,C 90.000,E1 296.309} C_DIS
LIN {X -0.009,Y -542.442,Z 1078.445,A 0.000,B 0.000,C 90.000,E1 296.027} C_DIS
LIN {X -0.152,Y -542.043,Z 1078.441,A 0.000,B 0.000,C 90.000,E1 295.335} C_DIS
LIN {X 0.080,Y -541.498,Z 1078.439,A 0.000,B 0.000,C 90.000,E1 295.027} C_DIS
LIN {X 0.086,Y -541.247,Z 1078.436,A 0.000,B 0.000,C 90.000,E1 294.463} C_DIS
LIN {X 0.022,Y -541.242,Z 1078.430,A 0.000,B 0.000,C 90.000,E1 293.334} C_DIS
LIN {X -0.085,Y -541.563,Z 1078.420,A 0.000,B 0.000,C 90.000,E1 291.642} C_DIS
LIN {X -0.317,Y -541.900,Z 1078.412,A 0.000,B 0.000,C 90.000,E1 290.248} C_DIS
LIN {X 0.157,Y -542.083,Z 1078.404,A 0.000,B 0.000,C 90.000,E1 288.779} C_DIS
LIN {X 0.223,Y -542.120,Z 1078.398,A 0.000,B 0.000,C 90.000,E1 287.638} C_DIS
LIN {X 0.290,Y -542.054,Z 1078.392,A 0.000,B 0.000,C 90.000,E1 286.496} C_DIS
LIN {X -0.245,Y -541.697,Z 1078.384,A 0.000,B 0.000,C 90.000,E1 285.134} C_DIS
LIN {X 0.195,Y -541.313,Z 1078.378,A 0.000,B 0.000,C 90.000,E1 283.953} C_DIS
LIN {X -0.276,Y -540.593,Z 1078.368,A 0.000,B 0.000,C 90.000,E1 282.299} C_DIS
LIN {X 0.172,Y -539.708,Z 1078.359,A 0.000,B 0.000,C 90.000,E1 280.546} C_DIS
LIN {X 0.101,Y -538.532,Z 1078.346,A 0.000,B 0.000,C 90.000,E1 278.276} C_DIS
LIN {X -0.224,Y -537.482,Z 1078.335,A 0.000,B 0.000,C 90.000,E1 276.315} C_DIS
LIN {X -0.088,Y -536.561,Z 1078.325,A 0.000,B 0.000,C 90.000,E1 274.588} C_DIS
LIN {X -0.048,Y -535.791,Z 1078.318,A 0.000,B 0.000,C 90.000,E1 273.154} C_DIS
LIN {X 0.004,Y -534.958,Z 1078.308,A 0.000,B 0.000,C 90.000,E1 271.432} C_DIS
LIN {X 0.005,Y -534.347,Z 1078.302,A 0.000,B 0.000,C 90.000,E1 270.286} C_DIS
LIN {X -0.001,Y -533.758,Z 1078.295,A 0.000,B 0.000,C 90.000,E1 269.141} C_DIS
LIN {X -0.017,Y -532.746,Z 1078.286,A 0.000,B 0.000,C 90.000,E1 267.421} C_DIS
LIN {X -0.026,Y -531.729,Z 1078.276,A 0.000,B 0.000,C 90.000,E1 265.698} C_DIS
LIN {X -0.038,Y -530.658,Z 1078.268,A 0.000,B 0.000,C 90.000,E1 264.261} C_DIS
LIN {X -0.019,Y -529.342,Z 1078.260,A 0.000,B 0.000,C 90.000,E1 262.818} C_DIS
LIN {X -0.002,Y -527.530,Z 1078.250,A 0.000,B 0.000,C 90.000,E1 261.084} C_DIS
LIN {X 0.050,Y -525.678,Z 1078.241,A 0.000,B 0.000,C 90.000,E1 259.342} C_DIS
LIN {X 0.166,Y -523.530,Z 1078.230,A 0.000,B 0.000,C 90.000,E1 257.297} C_DIS
LIN {X -0.186,Y -522.409,Z 1078.223,A 0.000,B 0.000,C 90.000,E1 256.172} C_DIS
LIN {X 0.083,Y -520.359,Z 1078.212,A 0.000,B 0.000,C 90.000,E1 254.102} C_DIS
LIN {X -0.048,Y -518.476,Z 1078.202,A 0.000,B 0.000,C 90.000,E1 252.362} C_DIS
LIN {X 0.166,Y -517.291,Z 1078.196,A 0.000,B 0.000,C 90.000,E1 251.167} C_DIS
LIN {X 0.169,Y -515.651,Z 1078.187,A 0.000,B 0.000,C 90.000,E1 249.699} C_DIS
LIN {X -0.209,Y -513.418,Z 1078.178,A 0.000,B 0.000,C 90.000,E1 247.975} C_DIS
LIN {X 0.031,Y -510.942,Z 1078.168,A 0.000,B 0.000,C 90.000,E1 246.177} C_DIS
LIN {X 0.209,Y -509.147,Z 1078.161,A 0.000,B 0.000,C 90.000,E1 244.973} C_DIS
LIN {X -0.002,Y -506.806,Z 1078.153,A 0.000,B 0.000,C 90.000,E1 243.512} C_DIS
LIN {X -0.028,Y -504.336,Z 1078.145,A 0.000,B 0.000,C 90.000,E1 242.025} C_DIS
LIN {X -0.105,Y -501.745,Z 1078.136,A 0.000,B 0.000,C 90.000,E1 240.539} C_DIS
LIN {X -0.032,Y -499.677,Z 1078.130,A 0.000,B 0.000,C 90.000,E1 239.331} C_DIS
LIN {X 0.300,Y -496.928,Z 1078.121,A 0.000,B 0.000,C 90.000,E1 237.788} C_DIS
LIN {X -0.115,Y -494.729,Z 1078.115,A 0.000,B 0.000,C 90.000,E1 236.628} C_DIS
LIN {X -0.025,Y -491.788,Z 1078.106,A 0.000,B 0.000,C 90.000,E1 235.102} C_DIS
LIN {X -0.235,Y -489.339,Z 1078.099,A 0.000,B 0.000,C 90.000,E1 233.909} C_DIS
LIN {X 0.196,Y -486.865,Z 1078.093,A 0.000,B 0.000,C 90.000,E1 232.637} C_DIS
LIN {X 0.017,Y -483.571,Z 1078.084,A 0.000,B 0.000,C 90.000,E1 231.126} C_DIS
LIN {X 0.016,Y -480.241,Z 1078.076,A 0.000,B 0.000,C 90.000,E1 229.585} C_DIS
LIN {X 0.007,Y -475.085,Z 1078.062,A 0.000,B 0.000,C 90.000,E1 227.106} C_DIS
LIN {X 0.021,Y -470.994,Z 1078.050,A 0.000,B 0.000,C 90.000,E1 224.919} C_DIS
LIN {X 0.196,Y -467.508,Z 1078.039,A 0.000,B 0.000,C 90.000,E1 223.014} C_DIS
LIN {X 0.158,Y -465.098,Z 1078.032,A 0.000,B 0.000,C 90.000,E1 221.757} C_DIS
LIN {X -0.079,Y -461.373,Z 1078.022,A 0.000,B 0.000,C 90.000,E1 219.886} C_DIS
LIN {X -0.139,Y -458.322,Z 1078.013,A 0.000,B 0.000,C 90.000,E1 218.302} C_DIS
LIN {X -0.099,Y -454.552,Z 1078.002,A 0.000,B 0.000,C 90.000,E1 216.377} C_DIS
LIN {X 0.224,Y -450.689,Z 1077.991,A 0.000,B 0.000,C 90.000,E1 214.405} C_DIS
LIN {X 0.261,Y -446.346,Z 1077.979,A 0.000,B 0.000,C 90.000,E1 212.133} C_DIS
LIN {X -0.025,Y -443.355,Z 1077.970,A 0.000,B 0.000,C 90.000,E1 210.541} C_DIS
LIN {X 0.068,Y -439.742,Z 1077.959,A 0.000,B 0.000,C 90.000,E1 208.565} C_DIS
LIN {X 0.100,Y -435.125,Z 1077.944,A 0.000,B 0.000,C 90.000,E1 205.924} C_DIS
LIN {X -0.022,Y -432.043,Z 1077.933,A 0.000,B 0.000,C 90.000,E1 203.951} C_DIS
LIN {X 0.213,Y -428.133,Z 1077.916,A 0.000,B 0.000,C 90.000,E1 200.918} C_DIS
LIN {X 0.024,Y -427.266,Z 1077.911,A 0.000,B 0.000,C 90.000,E1 199.939} C_DIS
LIN {X -0.177,Y -427.022,Z 1077.905,A 0.000,B 0.000,C 90.000,E1 198.960} C_DIS
LIN {X 0.224,Y -427.175,Z 1077.901,A 0.000,B 0.000,C 90.000,E1 198.236} C_DIS
LIN {X 0.089,Y -427.658,Z 1077.898,A 0.000,B 0.000,C 90.000,E1 197.583} C_DIS
LIN {X 0.086,Y -428.659,Z 1077.894,A 0.000,B 0.000,C 90.000,E1 196.913} C_DIS
LIN {X 0.174,Y -431.115,Z 1077.889,A 0.000,B 0.000,C 90.000,E1 195.898} C_DIS
LIN {X 0.180,Y -433.887,Z 1077.884,A 0.000,B 0.000,C 90.000,E1 195.064} C_DIS
LIN {X -0.081,Y -438.797,Z 1077.877,A 0.000,B 0.000,C 90.000,E1 193.939} C_DIS
LIN {X -0.217,Y -445.646,Z 1077.869,A 0.000,B 0.000,C 90.000,E1 192.479} C_DIS
LIN {X 0.137,Y -455.743,Z 1077.858,A 0.000,B 0.000,C 90.000,E1 190.489} C_DIS
LIN {X 0.199,Y -466.379,Z 1077.848,A 0.000,B 0.000,C 90.000,E1 188.568} C_DIS
LIN {X 0.129,Y -475.161,Z 1077.839,A 0.000,B 0.000,C 90.000,E1 187.004} C_DIS
LIN {X -0.006,Y -480.224,Z 1077.834,A 0.000,B 0.000,C 90.000,E1 186.087} C_DIS
LIN {X 0.126,Y -488.414,Z 1077.825,A 0.000,B 0.000,C 90.000,E1 184.531} C_DIS
LIN {X 0.167,Y -495.537,Z 1077.818,A 0.000,B 0.000,C 90.000,E1 183.154} C_DIS
LIN {X -0.160,Y -502.618,Z 1077.810,A 0.000,B 0.000,C 90.000,E1 181.835} C_DIS
LIN {X -0.081,Y -508.749,Z 1077.803,A 0.000,B 0.000,C 90.000,E1 180.630} C_DIS
LIN {X -0.215,Y -515.633,Z 1077.796,A 0.000,B 0.000,C 90.000,E1 179.312} C_DIS
LIN {X -0.186,Y -520.977,Z 1077.790,A 0.000,B 0.000,C 90.000,E1 178.282} C_DIS
LIN {X -0.143,Y -530.664,Z 1077.780,A 0.000,B 0.000,C 90.000,E1 176.388} C_DIS
LIN {X 0.186,Y -540.268,Z 1077.770,A 0.000,B 0.000,C 90.000,E1 174.489} C_DIS
LIN {X -0.173,Y -547.495,Z 1077.762,A 0.000,B 0.000,C 90.000,E1 173.109} C_DIS
LIN {X 0.274,Y -554.622,Z 1077.754,A 0.000,B 0.000,C 90.000,E1 171.659} C_DIS
LIN {X 0.223,Y -561.644,Z 1077.746,A 0.000,B 0.000,C 90.000,E1 170.274} C_DIS
LIN {X -0.074,Y -568.383,Z 1077.739,A 0.000,B 0.000,C 90.000,E1 168.926} C_DIS
LIN {X -0.006,Y -573.521,Z 1077.732,A 0.000,B 0.000,C 90.000,E1 167.825} C_DIS
LIN {X 0.252,Y -580.945,Z 1077.723,A 0.000,B 0.000,C 90.000,E1 166.172} C_DIS
LIN {X 0.277,Y -585.094,Z 1077.718,A 0.000,B 0.000,C 90.000,E1 165.227} C_DIS
LIN {X 0.017,Y -588.460,Z 1077.714,A 0.000,B 0.000,C 90.000,E1 164.448} C_DIS
LIN {X 0.052,Y -592.738,Z 1077.708,A 0.000,B 0.000,C 90.000,E1 163.378} C_DIS
LIN {X 0.139,Y -596.757,Z 1077.702,A 0.000,B 0.000,C 90.000,E1 162.308} C_DIS
LIN {X -0.109,Y -600.601,Z 1077.696,A 0.000,B 0.000,C 90.000,E1 161.275} C_DIS
LIN {X 0.187,Y -605.048,Z 1077.689,A 0.000,B 0.000,C 90.000,E1 159.934} C_DIS
LIN {X -0.006,Y -609.182,Z 1077.681,A 0.000,B 0.000,C 90.000,E1 158.646} C_DIS
LIN {X -0.174,Y -613.865,Z 1077.673,A 0.000,B 0.000,C 90.000,E1 157.102} C_DIS
LIN {X 0.030,Y -616.794,Z 1077.667,A 0.000,B 0.000,C 90.000,E1 156.049} C_DIS
LIN {X -0.327,Y -621.516,Z 1077.657,A 0.000,B 0.000,C 90.000,E1 154.280} C_DIS
LIN {X -0.327,Y -624.114,Z 1077.651,A 0.000,B 0.000,C 90.000,E1 153.256} C_DIS
LIN {X -0.280,Y -627.220,Z 1077.644,A 0.000,B 0.000,C 90.000,E1 151.975} C_DIS
LIN {X 0.111,Y -630.192,Z 1077.637,A 0.000,B 0.000,C 90.000,E1 150.667} C_DIS
LIN {X 0.032,Y -633.583,Z 1077.629,A 0.000,B 0.000,C 90.000,E1 149.154} C_DIS
LIN {X -0.198,Y -636.839,Z 1077.620,A 0.000,B 0.000,C 90.000,E1 147.661} C_DIS
LIN {X 0.030,Y -640.460,Z 1077.610,A 0.000,B 0.000,C 90.000,E1 145.881} C_DIS
LIN {X 0.180,Y -643.945,Z 1077.601,A 0.000,B 0.000,C 90.000,E1 144.116} C_DIS
LIN {X 0.324,Y -647.826,Z 1077.590,A 0.000,B 0.000,C 90.000,E1 142.110} C_DIS
LIN {X 0.086,Y -650.756,Z 1077.581,A 0.000,B 0.000,C 90.000,E1 140.642} C_DIS
LIN {X -0.106,Y -653.730,Z 1077.573,A 0.000,B 0.000,C 90.000,E1 139.175} C_DIS
LIN {X 0.126,Y -656.826,Z 1077.565,A 0.000,B 0.000,C 90.000,E1 137.676} C_DIS
LIN {X -0.082,Y -661.584,Z 1077.553,A 0.000,B 0.000,C 90.000,E1 135.486} C_DIS
LIN {X -0.156,Y -665.159,Z 1077.545,A 0.000,B 0.000,C 90.000,E1 134.028} C_DIS
LIN {X -0.131,Y -669.508,Z 1077.535,A 0.000,B 0.000,C 90.000,E1 132.324} C_DIS
LIN {X -0.018,Y -673.235,Z 1077.527,A 0.000,B 0.000,C 90.000,E1 130.862} C_DIS
LIN {X 0.138,Y -676.345,Z 1077.520,A 0.000,B 0.000,C 90.000,E1 129.644} C_DIS
LIN {X 0.064,Y -680.578,Z 1077.511,A 0.000,B 0.000,C 90.000,E1 127.971} C_DIS
LIN {X -0.104,Y -683.707,Z 1077.504,A 0.000,B 0.000,C 90.000,E1 126.790} C_DIS
LIN {X 0.286,Y -686.212,Z 1077.499,A 0.000,B 0.000,C 90.000,E1 125.804} C_DIS
LIN {X -0.022,Y -689.651,Z 1077.491,A 0.000,B 0.000,C 90.000,E1 124.405} C_DIS
LIN {X 0.306,Y -693.125,Z 1077.483,A 0.000,B 0.000,C 90.000,E1 122.959} C_DIS
LIN {X 0.085,Y -695.925,Z 1077.477,A 0.000,B 0.000,C 90.000,E1 121.799} C_DIS
LIN {X -0.115,Y -698.075,Z 1077.472,A 0.000,B 0.000,C 90.000,E1 120.875} C_DIS
LIN {X 0.411,Y -699.561,Z 1077.468,A 0.000,B 0.000,C 90.000,E1 120.129} C_DIS
LIN {X -0.011,Y -700.716,Z 1077.464,A 0.000,B 0.000,C 90.000,E1 119.461} C_DIS
LIN {X 0.187,Y -701.609,Z 1077.460,A 0.000,B 0.000,C 90.000,E1 118.743} C_DIS
LIN {X 0.221,Y -703.416,Z 1077.449,A 0.000,B 0.000,C 90.000,E1 116.873} C_DIS
LIN {X 0.069,Y -704.523,Z 1077.443,A 0.000,B 0.000,C 90.000,E1 115.720} C_DIS
LIN {X -0.298,Y -704.915,Z 1077.440,A 0.000,B 0.000,C 90.000,E1 115.283} C_DIS
LIN {X 0.278,Y -705.053,Z 1077.438,A 0.000,B 0.000,C 90.000,E1 114.771} C_DIS
LIN {X -0.076,Y -705.018,Z 1077.437,A 0.000,B 0.000,C 90.000,E1 114.567} C_DIS
LIN {X 0.205,Y -704.555,Z 1077.434,A 0.000,B 0.000,C 90.000,E1 114.079} C_DIS
LIN {X -0.154,Y -704.005,Z 1077.433,A 0.000,B 0.000,C 90.000,E1 113.875} C_DIS
LIN {X 0.126,Y -702.406,Z 1077.430,A 0.000,B 0.000,C 90.000,E1 113.387} C_DIS
LIN {X 0.264,Y -701.779,Z 1077.429,A 0.000,B 0.000,C 90.000,E1 113.259} C_DIS
LIN {X -0.114,Y -698.202,Z 1077.427,A 0.000,B 0.000,C 90.000,E1 112.823} C_DIS
LIN {X 0.016,Y -697.125,Z 1077.426,A 0.000,B 0.000,C 90.000,E1 112.695} C_DIS
LIN {X -0.123,Y -695.487,Z 1077.426,A 0.000,B 0.000,C 90.000,E1 112.589} C_DIS
LIN {X 0.399,Y -687.990,Z 1077.424,A 0.000,B 0.000,C 90.000,E1 112.206} C_DIS
LIN {X 0.171,Y -686.111,Z 1077.423,A 0.000,B 0.000,C 90.000,E1 112.153} C_DIS
LIN {X 0.105,Y -683.457,Z 1077.423,A 0.000,B 0.000,C 90.000,E1 112.099} C_DIS
LIN {X -0.122,Y -676.141,Z 1077.422,A 0.000,B 0.000,C 90.000,E1 112.025} C_DIS
LIN {X -0.157,Y -606.314,Z 1077.422,A 0.000,B 0.000,C 90.000,E1 112.025} C_DIS
LIN {X 0.081,Y -602.667,Z 1077.422,A 0.000,B 0.000,C 90.000,E1 111.844} C_DIS
LIN {X -0.327,Y -599.754,Z 1077.421,A 0.000,B 0.000,C 90.000,E1 111.716} C_DIS
LIN {X 0.131,Y -596.715,Z 1077.419,A 0.000,B 0.000,C 90.000,E1 111.482} C_DIS
LIN {X 0.105,Y -589.463,Z 1077.416,A 0.000,B 0.000,C 90.000,E1 110.918} C_DIS
LIN {X 0.019,Y -578.352,Z 1077.411,A 0.000,B 0.000,C 90.000,E1 109.993} C_DIS
LIN {X 0.108,Y -573.950,Z 1077.409,A 0.000,B 0.000,C 90.000,E1 109.631} C_DIS
LIN {X -0.112,Y -567.869,Z 1077.407,A 0.000,B 0.000,C 90.000,E1 109.214} C_DIS
LIN {X 0.289,Y -561.515,Z 1077.405,A 0.000,B 0.000,C 90.000,E1 108.779} C_DIS
LIN {X -0.037,Y -553.629,Z 1077.402,A 0.000,B 0.000,C 90.000,E1 108.362} C_DIS
LIN {X 0.121,Y -549.419,Z 1077.400,A 0.000,B 0.000,C 90.000,E1 108.055} C_DIS
LIN {X -0.113,Y -547.745,Z 1077.399,A 0.000,B 0.000,C 90.000,E1 107.873} C_DIS
LIN {X -0.155,Y -547.722,Z 1077.399,A 0.000,B 0.000,C 90.000,E1 107.873} C_DIS
LIN {X 0.242,Y -547.351,Z 1077.397,A 0.000,B 0.000,C 90.000,E1 107.511} C_DIS
LIN {X -0.006,Y -548.606,Z 1077.386,A 0.000,B 0.000,C 90.000,E1 105.426} C_DIS
LIN {X 0.026,Y -550.265,Z 1077.373,A 0.000,B 0.000,C 90.000,E1 103.175} C_DIS
LIN {X -0.148,Y -552.240,Z 1077.361,A 0.000,B 0.000,C 90.000,E1 100.950} C_DIS
LIN {X 0.051,Y -554.291,Z 1077.350,A 0.000,B 0.000,C 90.000,E1 98.973} C_DIS
LIN {X -0.037,Y -555.850,Z 1077.342,A 0.000,B 0.000,C 90.000,E1 97.587} C_DIS
LIN {X -0.092,Y -557.393,Z 1077.334,A 0.000,B 0.000,C 90.000,E1 96.201} C_DIS
LIN {X -0.177,Y -558.820,Z 1077.327,A 0.000,B 0.000,C 90.000,E1 94.821} C_DIS
LIN {X 0.234,Y -559.634,Z 1077.321,A 0.000,B 0.000,C 90.000,E1 93.669} C_DIS
LIN {X 0.148,Y -560.430,Z 1077.313,A 0.000,B 0.000,C 90.000,E1 92.293} C_DIS
LIN {X 0.075,Y -561.139,Z 1077.305,A 0.000,B 0.000,C 90.000,E1 90.917} C_DIS
LIN {X -0.097,Y -561.615,Z 1077.299,A 0.000,B 0.000,C 90.000,E1 89.828} C_DIS
LIN {X -0.049,Y -562.250,Z 1077.290,A 0.000,B 0.000,C 90.000,E1 88.165} C_DIS
LIN {X -0.084,Y -562.790,Z 1077.282,A 0.000,B 0.000,C 90.000,E1 86.788} C_DIS
LIN {X -0.119,Y -563.339,Z 1077.275,A 0.000,B 0.000,C 90.000,E1 85.412} C_DIS
LIN {X 0.039,Y -563.873,Z 1077.265,A 0.000,B 0.000,C 90.000,E1 83.742} C_DIS
LIN {X -0.196,Y -564.468,Z 1077.255,A 0.000,B 0.000,C 90.000,E1 81.837} C_DIS
LIN {X -0.181,Y -565.236,Z 1077.242,A 0.000,B 0.000,C 90.000,E1 79.634} C_DIS
LIN {X 0.108,Y -565.866,Z 1077.235,A 0.000,B 0.000,C 90.000,E1 78.229} C_DIS
LIN {X 0.125,Y -567.174,Z 1077.221,A 0.000,B 0.000,C 90.000,E1 75.755} C_DIS
LIN {X 0.277,Y -569.311,Z 1077.204,A 0.000,B 0.000,C 90.000,E1 72.725} C_DIS
LIN {X 0.174,Y -570.626,Z 1077.195,A 0.000,B 0.000,C 90.000,E1 71.094} C_DIS
LIN {X -0.088,Y -572.244,Z 1077.184,A 0.000,B 0.000,C 90.000,E1 69.209} C_DIS
LIN {X 0.103,Y -573.811,Z 1077.174,A 0.000,B 0.000,C 90.000,E1 67.283} C_DIS
LIN {X -0.032,Y -575.089,Z 1077.165,A 0.000,B 0.000,C 90.000,E1 65.665} C_DIS
LIN {X 0.239,Y -575.979,Z 1077.157,A 0.000,B 0.000,C 90.000,E1 64.280} C_DIS
LIN {X -0.002,Y -576.761,Z 1077.150,A 0.000,B 0.000,C 90.000,E1 62.948} C_DIS
LIN {X -0.183,Y -577.265,Z 1077.145,A 0.000,B 0.000,C 90.000,E1 62.153} C_DIS
LIN {X -0.004,Y -578.214,Z 1077.136,A 0.000,B 0.000,C 90.000,E1 60.511} C_DIS
LIN {X 0.044,Y -578.861,Z 1077.129,A 0.000,B 0.000,C 90.000,E1 59.154} C_DIS
LIN {X 0.039,Y -579.413,Z 1077.123,A 0.000,B 0.000,C 90.000,E1 58.074} C_DIS
LIN {X 0.366,Y -580.149,Z 1077.114,A 0.000,B 0.000,C 90.000,E1 56.421} C_DIS
LIN {X -0.100,Y -580.859,Z 1077.105,A 0.000,B 0.000,C 90.000,E1 54.848} C_DIS
LIN {X -0.060,Y -581.230,Z 1077.097,A 0.000,B 0.000,C 90.000,E1 53.497} C_DIS
LIN {X 0.168,Y -581.436,Z 1077.091,A 0.000,B 0.000,C 90.000,E1 52.396} C_DIS
LIN {X -0.129,Y -581.461,Z 1077.087,A 0.000,B 0.000,C 90.000,E1 51.618} C_DIS
LIN {X -0.067,Y -581.363,Z 1077.082,A 0.000,B 0.000,C 90.000,E1 50.803} C_DIS
LIN {X 0.050,Y -580.893,Z 1077.073,A 0.000,B 0.000,C 90.000,E1 49.175} C_DIS
LIN {X 0.209,Y -580.463,Z 1077.067,A 0.000,B 0.000,C 90.000,E1 48.081} C_DIS
LIN {X 0.098,Y -579.777,Z 1077.060,A 0.000,B 0.000,C 90.000,E1 46.743} C_DIS
LIN {X 0.247,Y -579.059,Z 1077.054,A 0.000,B 0.000,C 90.000,E1 45.648} C_DIS
LIN {X -0.030,Y -578.122,Z 1077.048,A 0.000,B 0.000,C 90.000,E1 44.595} C_DIS
LIN {X 0.095,Y -576.926,Z 1077.042,A 0.000,B 0.000,C 90.000,E1 43.500} C_DIS
LIN {X -0.078,Y -575.093,Z 1077.034,A 0.000,B 0.000,C 90.000,E1 42.162} C_DIS
LIN {X -0.137,Y -573.903,Z 1077.030,A 0.000,B 0.000,C 90.000,E1 41.353} C_DIS
LIN {X -0.024,Y -571.882,Z 1077.024,A 0.000,B 0.000,C 90.000,E1 40.253} C_DIS
LIN {X 0.073,Y -569.605,Z 1077.018,A 0.000,B 0.000,C 90.000,E1 39.152} C_DIS
LIN {X 0.015,Y -567.655,Z 1077.013,A 0.000,B 0.000,C 90.000,E1 38.338} C_DIS
LIN {X -0.185,Y -566.262,Z 1077.010,A 0.000,B 0.000,C 90.000,E1 37.810} C_DIS
LIN {X 0.050,Y -564.695,Z 1077.007,A 0.000,B 0.000,C 90.000,E1 37.237} C_DIS
LIN {X -0.071,Y -562.040,Z 1077.002,A 0.000,B 0.000,C 90.000,E1 36.423} C_DIS
LIN {X -0.199,Y -560.192,Z 1076.999,A 0.000,B 0.000,C 90.000,E1 35.884} C_DIS
LIN {X -0.008,Y -558.061,Z 1076.996,A 0.000,B 0.000,C 90.000,E1 35.311} C_DIS
LIN {X 0.002,Y -553.283,Z 1076.990,A 0.000,B 0.000,C 90.000,E1 34.199} C_DIS
LIN {X -0.116,Y -549.416,Z 1076.985,A 0.000,B 0.000,C 90.000,E1 33.372} C_DIS
LIN {X 0.345,Y -544.489,Z 1076.980,A 0.000,B 0.000,C 90.000,E1 32.339} C_DIS
LIN {X -0.160,Y -539.887,Z 1076.975,A 0.000,B 0.000,C 90.000,E1 31.544} C_DIS
LIN {X 0.033,Y -535.023,Z 1076.970,A 0.000,B 0.000,C 90.000,E1 30.669} C_DIS
LIN {X 0.048,Y -530.626,Z 1076.966,A 0.000,B 0.000,C 90.000,E1 29.951} C_DIS
LIN {X 0.282,Y -525.659,Z 1076.963,A 0.000,B 0.000,C 90.000,E1 29.205} C_DIS
LIN {X 0.210,Y -520.334,Z 1076.958,A 0.000,B 0.000,C 90.000,E1 28.487} C_DIS
LIN {X 0.088,Y -514.703,Z 1076.954,A 0.000,B 0.000,C 90.000,E1 27.769} C_DIS
LIN {X -0.082,Y -508.460,Z 1076.950,A 0.000,B 0.000,C 90.000,E1 27.052} C_DIS
LIN {X -0.253,Y -503.175,Z 1076.947,A 0.000,B 0.000,C 90.000,E1 26.488} C_DIS
LIN {X 0.134,Y -495.095,Z 1076.942,A 0.000,B 0.000,C 90.000,E1 25.591} C_DIS
LIN {X -0.070,Y -484.074,Z 1076.936,A 0.000,B 0.000,C 90.000,E1 24.515} C_DIS
LIN {X -0.108,Y -473.962,Z 1076.931,A 0.000,B 0.000,C 90.000,E1 23.567} C_DIS
LIN {X 0.099,Y -462.201,Z 1076.925,A 0.000,B 0.000,C 90.000,E1 22.514} C_DIS
LIN {X -0.168,Y -444.212,Z 1076.916,A 0.000,B 0.000,C 90.000,E1 20.972} C_DIS
LIN {X 0.030,Y -429.482,Z 1076.909,A 0.000,B 0.000,C 90.000,E1 19.577} C_DIS
LIN {X 0.109,Y -416.638,Z 1076.901,A 0.000,B 0.000,C 90.000,E1 18.236} C_DIS
LIN {X -0.034,Y -405.720,Z 1076.894,A 0.000,B 0.000,C 90.000,E1 16.985} C_DIS
LIN {X 0.152,Y -399.404,Z 1076.890,A 0.000,B 0.000,C 90.000,E1 16.134} C_DIS
LIN {X 0.111,Y -396.366,Z 1076.887,A 0.000,B 0.000,C 90.000,E1 15.662} C_DIS
LIN {X 0.138,Y -393.228,Z 1076.883,A 0.000,B 0.000,C 90.000,E1 14.954} C_DIS
LIN {X -0.019,Y -392.297,Z 1076.881,A 0.000,B 0.000,C 90.000,E1 14.537} C_DIS
LIN {X -0.025,Y -391.835,Z 1076.877,A 0.000,B 0.000,C 90.000,E1 13.828} C_DIS
LIN {X -0.036,Y -392.371,Z 1076.873,A 0.000,B 0.000,C 90.000,E1 13.119} C_DIS
LIN {X -0.135,Y -395.341,Z 1076.861,A 0.000,B 0.000,C 90.000,E1 11.007} C_DIS
LIN {X 0.043,Y -400.335,Z 1076.845,A 0.000,B 0.000,C 90.000,E1 8.163} C_DIS
LIN {X -0.110,Y -404.851,Z 1076.834,A 0.000,B 0.000,C 90.000,E1 6.087} C_DIS
LIN {X -0.148,Y -407.043,Z 1076.828,A 0.000,B 0.000,C 90.000,E1 5.049} C_DIS
LIN {X -0.170,Y -408.926,Z 1076.824,A 0.000,B 0.000,C 90.000,E1 4.359} C_DIS
LIN {X -0.163,Y -410.295,Z 1076.822,A 0.000,B 0.000,C 90.000,E1 4.012} C_DIS
LIN {X 0.025,Y -412.302,Z 1076.820,A 0.000,B 0.000,C 90.000,E1 3.555} C_DIS
LIN {X -0.070,Y -417.061,Z 1076.817,A 0.000,B 0.000,C 90.000,E1 2.980} C_DIS
LIN {X -0.056,Y -421.333,Z 1076.815,A 0.000,B 0.000,C 90.000,E1 2.636} C_DIS
LIN {X 0.047,Y -431.561,Z 1076.811,A 0.000,B 0.000,C 90.000,E1 1.949} C_DIS
LIN {X -0.027,Y -454.712,Z 1076.803,A 0.000,B 0.000,C 90.000,E1 0.458} C_DIS
LIN {X 0.156,Y -471.945,Z 1076.797,A 0.000,B 0.000,C 90.000,E1 359.370} C_DIS
LIN {X 0.090,Y -484.977,Z 1076.792,A 0.000,B 0.000,C 90.000,E1 358.568} C_DIS
LIN {X 0.099,Y -494.652,Z 1076.789,A 0.000,B 0.000,C 90.000,E1 357.936} C_DIS
LIN {X -0.043,Y -504.028,Z 1076.785,A 0.000,B 0.000,C 90.000,E1 357.306} C_DIS
LIN {X -0.230,Y -511.417,Z 1076.782,A 0.000,B 0.000,C 90.000,E1 356.788} C_DIS
LIN {X -0.227,Y -517.293,Z 1076.780,A 0.000,B 0.000,C 90.000,E1 356.331} C_DIS
LIN {X 0.141,Y -524.317,Z 1076.776,A 0.000,B 0.000,C 90.000,E1 355.698} C_DIS
LIN {X -0.169,Y -532.532,Z 1076.772,A 0.000,B 0.000,C 90.000,E1 354.951} C_DIS
LIN {X 0.113,Y -537.753,Z 1076.769,A 0.000,B 0.000,C 90.000,E1 354.375} C_DIS
LIN {X -0.008,Y -543.825,Z 1076.765,A 0.000,B 0.000,C 90.000,E1 353.685} C_DIS
LIN {X 0.099,Y -548.410,Z 1076.762,A 0.000,B 0.000,C 90.000,E1 353.109} C_DIS
LIN {X 0.055,Y -553.374,Z 1076.758,A 0.000,B 0.000,C 90.000,E1 352.413} C_DIS
LIN {X 0.217,Y -557.009,Z 1076.755,A 0.000,B 0.000,C 90.000,E1 351.837} C_DIS
LIN {X 0.240,Y -561.058,Z 1076.751,A 0.000,B 0.000,C 90.000,E1 351.141} C_DIS
LIN {X -0.257,Y -564.747,Z 1076.747,A 0.000,B 0.000,C 90.000,E1 350.500} C_DIS
LIN {X 0.151,Y -568.734,Z 1076.743,A 0.000,B 0.000,C 90.000,E1 349.634} C_DIS
LIN {X 0.142,Y -572.289,Z 1076.738,A 0.000,B 0.000,C 90.000,E1 348.814} C_DIS
LIN {X -0.031,Y -574.645,Z 1076.735,A 0.000,B 0.000,C 90.000,E1 348.285} C_DIS
LIN {X 0.237,Y -578.947,Z 1076.729,A 0.000,B 0.000,C 90.000,E1 347.173} C_DIS
LIN {X -0.006,Y -582.957,Z 1076.723,A 0.000,B 0.000,C 90.000,E1 346.117} C_DIS
LIN {X 0.188,Y -587.679,Z 1076.715,A 0.000,B 0.000,C 90.000,E1 344.755} C_DIS
LIN {X -0.045,Y -590.355,Z 1076.711,A 0.000,B 0.000,C 90.000,E1 343.976} C_DIS
LIN {X -0.122,Y -594.699,Z 1076.704,A 0.000,B 0.000,C 90.000,E1 342.653} C_DIS
LIN {X -0.012,Y -598.018,Z 1076.698,A 0.000,B 0.000,C 90.000,E1 341.583} C_DIS
LIN {X 0.051,Y -600.303,Z 1076.693,A 0.000,B 0.000,C 90.000,E1 340.786} C_DIS
LIN {X 0.051,Y -604.427,Z 1076.685,A 0.000,B 0.000,C 90.000,E1 339.209} C_DIS
LIN {X 0.187,Y -606.301,Z 1076.680,A 0.000,B 0.000,C 90.000,E1 338.411} C_DIS
LIN {X -0.055,Y -609.554,Z 1076.672,A 0.000,B 0.000,C 90.000,E1 336.869} C_DIS
LIN {X 0.328,Y -611.342,Z 1076.666,A 0.000,B 0.000,C 90.000,E1 335.793} C_DIS
LIN {X -0.037,Y -612.510,Z 1076.661,A 0.000,B 0.000,C 90.000,E1 335.049} C_DIS
LIN {X -0.162,Y -613.973,Z 1076.656,A 0.000,B 0.000,C 90.000,E1 334.024} C_DIS
LIN {X -0.264,Y -615.234,Z 1076.650,A 0.000,B 0.000,C 90.000,E1 332.999} C_DIS
LIN {X -0.332,Y -616.048,Z 1076.646,A 0.000,B 0.000,C 90.000,E1 332.231} C_DIS
LIN {X -0.121,Y -616.991,Z 1076.640,A 0.000,B 0.000,C 90.000,E1 331.179} C_DIS
LIN {X 0.126,Y -617.478,Z 1076.636,A 0.000,B 0.000,C 90.000,E1 330.383} C_DIS
LIN {X 0.362,Y -617.806,Z 1076.630,A 0.000,B 0.000,C 90.000,E1 329.331} C_DIS
LIN {X 0.067,Y -617.883,Z 1076.624,A 0.000,B 0.000,C 90.000,E1 328.329} C_DIS
LIN {X 0.071,Y -617.488,Z 1076.617,A 0.000,B 0.000,C 90.000,E1 327.041} C_DIS
LIN {X 0.099,Y -616.793,Z 1076.611,A 0.000,B 0.000,C 90.000,E1 326.008} C_DIS
LIN {X 0.116,Y -615.866,Z 1076.605,A 0.000,B 0.000,C 90.000,E1 324.975} C_DIS
LIN {X -0.344,Y -614.085,Z 1076.595,A 0.000,B 0.000,C 90.000,E1 323.210} C_DIS
LIN {X -0.099,Y -612.474,Z 1076.585,A 0.000,B 0.000,C 90.000,E1 321.376} C_DIS
LIN {X -0.074,Y -610.870,Z 1076.574,A 0.000,B 0.000,C 90.000,E1 319.299} C_DIS
LIN {X 0.114,Y -610.195,Z 1076.568,A 0.000,B 0.000,C 90.000,E1 318.243} C_DIS
LIN {X 0.203,Y -609.790,Z 1076.565,A 0.000,B 0.000,C 90.000,E1 317.715} C_DIS
LIN {X 0.020,Y -609.658,Z 1076.564,A 0.000,B 0.000,C 90.000,E1 317.472} C_DIS
LIN {X 0.228,Y -608.102,Z 1076.555,A 0.000,B 0.000,C 90.000,E1 315.891} C_DIS
LIN {X -0.031,Y -606.517,Z 1076.546,A 0.000,B 0.000,C 90.000,E1 314.352} C_DIS
LIN {X -0.220,Y -606.217,Z 1076.545,A 0.000,B 0.000,C 90.000,E1 314.109} C_DIS
LIN {X 0.107,Y -605.682,Z 1076.541,A 0.000,B 0.000,C 90.000,E1 313.299} C_DIS
LIN {X -0.231,Y -604.769,Z 1076.535,A 0.000,B 0.000,C 90.000,E1 312.285} C_DIS
LIN {X 0.248,Y -601.888,Z 1076.519,A 0.000,B 0.000,C 90.000,E1 309.358} C_DIS
LIN {X -0.031,Y -599.734,Z 1076.507,A 0.000,B 0.000,C 90.000,E1 307.282} C_DIS
LIN {X -0.018,Y -598.240,Z 1076.500,A 0.000,B 0.000,C 90.000,E1 305.964} C_DIS
LIN {X 0.094,Y -596.715,Z 1076.494,A 0.000,B 0.000,C 90.000,E1 304.898} C_DIS
LIN {X -0.048,Y -595.273,Z 1076.490,A 0.000,B 0.000,C 90.000,E1 304.119} C_DIS
LIN {X 0.066,Y -594.499,Z 1076.487,A 0.000,B 0.000,C 90.000,E1 303.579} C_DIS
LIN {X 0.177,Y -593.461,Z 1076.484,A 0.000,B 0.000,C 90.000,E1 303.038} C_DIS
LIN {X -0.107,Y -592.872,Z 1076.482,A 0.000,B 0.000,C 90.000,E1 302.801} C_DIS
LIN {X -0.217,Y -592.485,Z 1076.481,A 0.000,B 0.000,C 90.000,E1 302.546} C_DIS
LIN {X -0.120,Y -591.274,Z 1076.478,A 0.000,B 0.000,C 90.000,E1 302.005} C_DIS
LIN {X 0.081,Y -590.525,Z 1076.476,A 0.000,B 0.000,C 90.000,E1 301.720} C_DIS
LIN {X 0.047,Y -587.830,Z 1076.472,A 0.000,B 0.000,C 90.000,E1 300.924} C_DIS
LIN {X -0.071,Y -586.692,Z 1076.470,A 0.000,B 0.000,C 90.000,E1 300.669} C_DIS
LIN {X -0.013,Y -584.763,Z 1076.467,A 0.000,B 0.000,C 90.000,E1 300.129} C_DIS
LIN {X -0.040,Y -581.711,Z 1076.464,A 0.000,B 0.000,C 90.000,E1 299.461} C_DIS
LIN {X -0.310,Y -578.960,Z 1076.461,A 0.000,B 0.000,C 90.000,E1 298.949} C_DIS
LIN {X 0.263,Y -576.374,Z 1076.458,A 0.000,B 0.000,C 90.000,E1 298.487} C_DIS
LIN {X -0.039,Y -572.312,Z 1076.455,A 0.000,B 0.000,C 90.000,E1 297.975} C_DIS
LIN {X -0.017,Y -568.660,Z 1076.453,A 0.000,B 0.000,C 90.000,E1 297.564} C_DIS
LIN {X -0.094,Y -565.924,Z 1076.452,A 0.000,B 0.000,C 90.000,E1 297.308} C_DIS
LIN {X 0.017,Y -562.742,Z 1076.450,A 0.000,B 0.000,C 90.000,E1 297.052} C_DIS
LIN {X 0.120,Y -560.645,Z 1076.450,A 0.000,B 0.000,C 90.000,E1 296.924} C_DIS
LIN {X 0.088,Y -554.805,Z 1076.448,A 0.000,B 0.000,C 90.000,E1 296.668} C_DIS
LIN {X -0.173,Y -553.350,Z 1076.448,A 0.000,B 0.000,C 90.000,E1 296.616} C_DIS
LIN {X -0.277,Y -551.566,Z 1076.447,A 0.000,B 0.000,C 90.000,E1 296.488} C_DIS
LIN {X -0.008,Y -549.235,Z 1076.446,A 0.000,B 0.000,C 90.000,E1 296.232} C_DIS
LIN {X -0.157,Y -547.305,Z 1076.445,A 0.000,B 0.000,C 90.000,E1 296.027} C_DIS
LIN {X 0.217,Y -546.490,Z 1076.444,A 0.000,B 0.000,C 90.000,E1 295.848} C_DIS
LIN {X 0.098,Y -545.981,Z 1076.443,A 0.000,B 0.000,C 90.000,E1 295.720} C_DIS
LIN {X -0.024,Y -545.247,Z 1076.442,A 0.000,B 0.000,C 90.000,E1 295.591} C_DIS
LIN {X -0.146,Y -544.310,Z 1076.441,A 0.000,B 0.000,C 90.000,E1 295.463} C_DIS
LIN {X 0.097,Y -543.471,Z 1076.440,A 0.000,B 0.000,C 90.000,E1 295.155} C_DIS
LIN {X -0.157,Y -542.784,Z 1076.438,A 0.000,B 0.000,C 90.000,E1 294.899} C_DIS
LIN {X 0.122,Y -542.468,Z 1076.435,A 0.000,B 0.000,C 90.000,E1 294.335} C_DIS
LIN {X -0.137,Y -542.451,Z 1076.434,A 0.000,B 0.000,C 90.000,E1 294.079} C_DIS
LIN {X 0.099,Y -542.079,Z 1076.432,A 0.000,B 0.000,C 90.000,E1 293.770} C_DIS
LIN {X -0.068,Y -541.803,Z 1076.427,A 0.000,B 0.000,C 90.000,E1 292.950} C_DIS
LIN {X 0.166,Y -541.877,Z 1076.426,A 0.000,B 0.000,C 90.000,E1 292.642} C_DIS
LIN {X -0.132,Y -542.103,Z 1076.412,A 0.000,B 0.000,C 90.000,E1 290.120} C_DIS
LIN {X -0.114,Y -542.372,Z 1076.402,A 0.000,B 0.000,C 90.000,E1 288.417} C_DIS
LIN {X 0.023,Y -542.420,Z 1076.394,A 0.000,B 0.000,C 90.000,E1 286.985} C_DIS
LIN {X 0.169,Y -542.157,Z 1076.387,A 0.000,B 0.000,C 90.000,E1 285.552} C_DIS
LIN {X 0.302,Y -541.702,Z 1076.379,A 0.000,B 0.000,C 90.000,E1 284.120} C_DIS
LIN {X -0.288,Y -540.979,Z 1076.369,A 0.000,B 0.000,C 90.000,E1 282.479} C_DIS
LIN {X 0.203,Y -540.281,Z 1076.361,A 0.000,B 0.000,C 90.000,E1 281.007} C_DIS
LIN {X 0.007,Y -539.340,Z 1076.352,A 0.000,B 0.000,C 90.000,E1 279.321} C_DIS
LIN {X 0.256,Y -538.596,Z 1076.344,A 0.000,B 0.000,C 90.000,E1 277.871} C_DIS
LIN {X -0.122,Y -537.714,Z 1076.334,A 0.000,B 0.000,C 90.000,E1 276.201} C_DIS
LIN {X 0.023,Y -536.631,Z 1076.323,A 0.000,B 0.000,C 90.000,E1 274.188} C_DIS
LIN {X 0.103,Y -535.595,Z 1076.312,A 0.000,B 0.000,C 90.000,E1 272.178} C_DIS
LIN {X 0.129,Y -534.714,Z 1076.303,A 0.000,B 0.000,C 90.000,E1 270.458} C_DIS
LIN {X 0.128,Y -533.930,Z 1076.295,A 0.000,B 0.000,C 90.000,E1 269.026} C_DIS
LIN {X 0.121,Y -533.106,Z 1076.287,A 0.000,B 0.000,C 90.000,E1 267.593} C_DIS
LIN {X 0.122,Y -532.118,Z 1076.277,A 0.000,B 0.000,C 90.000,E1 265.869} C_DIS
LIN {X 0.119,Y -531.065,Z 1076.269,A 0.000,B 0.000,C 90.000,E1 264.432} C_DIS
LIN {X 0.085,Y -529.753,Z 1076.261,A 0.000,B 0.000,C 90.000,E1 262.996} C_DIS
LIN {X 0.155,Y -528.276,Z 1076.253,A 0.000,B 0.000,C 90.000,E1 261.546} C_DIS
LIN {X 0.252,Y -526.106,Z 1076.242,A 0.000,B 0.000,C 90.000,E1 259.511} C_DIS
LIN {X -0.123,Y -523.959,Z 1076.231,A 0.000,B 0.000,C 90.000,E1 257.521} C_DIS
LIN {X -0.068,Y -522.501,Z 1076.223,A 0.000,B 0.000,C 90.000,E1 256.061} C_DIS
LIN {X -0.164,Y -520.444,Z 1076.211,A 0.000,B 0.000,C 90.000,E1 254.031} C_DIS
LIN {X 0.213,Y -518.578,Z 1076.202,A 0.000,B 0.000,C 90.000,E1 252.236} C_DIS
LIN {X -0.058,Y -517.382,Z 1076.195,A 0.000,B 0.000,C 90.000,E1 251.094} C_DIS
LIN {X -0.045,Y -515.741,Z 1076.187,A 0.000,B 0.000,C 90.000,E1 249.625} C_DIS
LIN {X -0.060,Y -513.887,Z 1076.179,A 0.000,B 0.000,C 90.000,E1 248.156} C_DIS
LIN {X 0.193,Y -511.445,Z 1076.169,A 0.000,B 0.000,C 90.000,E1 246.357} C_DIS
LIN {X -0.191,Y -509.183,Z 1076.161,A 0.000,B 0.000,C 90.000,E1 244.921} C_DIS
LIN {X 0.275,Y -506.835,Z 1076.152,A 0.000,B 0.000,C 90.000,E1 243.384} C_DIS
LIN {X 0.248,Y -504.330,Z 1076.144,A 0.000,B 0.000,C 90.000,E1 241.897} C_DIS
LIN {X -0.270,Y -501.761,Z 1076.136,A 0.000,B 0.000,C 90.000,E1 240.461} C_DIS
LIN {X 0.136,Y -498.614,Z 1076.126,A 0.000,B 0.000,C 90.000,E1 238.614} C_DIS
LIN {X -0.123,Y -495.307,Z 1076.116,A 0.000,B 0.000,C 90.000,E1 236.834} C_DIS
LIN {X 0.232,Y -491.759,Z 1076.106,A 0.000,B 0.000,C 90.000,E1 234.975} C_DIS
LIN {X -0.142,Y -488.708,Z 1076.097,A 0.000,B 0.000,C 90.000,E1 233.497} C_DIS
LIN {X 0.018,Y -485.501,Z 1076.089,A 0.000,B 0.000,C 90.000,E1 231.949} C_DIS
LIN {X -0.244,Y -480.785,Z 1076.077,A 0.000,B 0.000,C 90.000,E1 229.828} C_DIS
LIN {X 0.084,Y -475.566,Z 1076.063,A 0.000,B 0.000,C 90.000,E1 227.310} C_DIS
LIN {X -0.120,Y -470.843,Z 1076.049,A 0.000,B 0.000,C 90.000,E1 224.838} C_DIS
LIN {X -0.024,Y -467.995,Z 1076.040,A 0.000,B 0.000,C 90.000,E1 223.257} C_DIS
LIN {X 0.013,Y -464.969,Z 1076.032,A 0.000,B 0.000,C 90.000,E1 221.676} C_DIS
LIN {X 0.066,Y -461.189,Z 1076.021,A 0.000,B 0.000,C 90.000,E1 219.769} C_DIS
LIN {X 0.067,Y -458.126,Z 1076.012,A 0.000,B 0.000,C 90.000,E1 218.177} C_DIS
LIN {X -0.259,Y -454.321,Z 1076.001,A 0.000,B 0.000,C 90.000,E1 216.297} C_DIS
LIN {X 0.055,Y -450.394,Z 1075.991,A 0.000,B 0.000,C 90.000,E1 214.326} C_DIS
LIN {X -0.156,Y -446.000,Z 1075.978,A 0.000,B 0.000,C 90.000,E1 212.084} C_DIS
LIN {X -0.215,Y -442.990,Z 1075.969,A 0.000,B 0.000,C 90.000,E1 210.463} C_DIS
LIN {X -0.177,Y -439.926,Z 1075.960,A 0.000,B 0.000,C 90.000,E1 208.821} C_DIS
LIN {X 0.052,Y -435.199,Z 1075.945,A 0.000,B 0.000,C 90.000,E1 206.155} C_DIS
LIN {X 0.132,Y -431.486,Z 1075.932,A 0.000,B 0.000,C 90.000,E1 203.823} C_DIS
LIN {X 0.160,Y -429.070,Z 1075.923,A 0.000,B 0.000,C 90.000,E1 202.153} C_DIS
LIN {X 0.141,Y -427.081,Z 1075.914,A 0.000,B 0.000,C 90.000,E1 200.482} C_DIS
LIN {X -0.062,Y -426.376,Z 1075.908,A 0.000,B 0.000,C 90.000,E1 199.504} C_DIS
LIN {X -0.070,Y -426.083,Z 1075.905,A 0.000,B 0.000,C 90.000,E1 198.833} C_DIS
LIN {X -0.217,Y -426.171,Z 1075.901,A 0.000,B 0.000,C 90.000,E1 198.181} C_DIS
LIN {X 0.178,Y -426.590,Z 1075.897,A 0.000,B 0.000,C 90.000,E1 197.457} C_DIS
LIN {X 0.042,Y -427.479,Z 1075.893,A 0.000,B 0.000,C 90.000,E1 196.804} C_DIS
LIN {X 0.118,Y -429.758,Z 1075.888,A 0.000,B 0.000,C 90.000,E1 195.788} C_DIS
LIN {X 0.114,Y -432.449,Z 1075.883,A 0.000,B 0.000,C 90.000,E1 194.954} C_DIS
LIN {X 0.137,Y -435.850,Z 1075.879,A 0.000,B 0.000,C 90.000,E1 194.120} C_DIS
LIN {X 0.052,Y -442.605,Z 1075.870,A 0.000,B 0.000,C 90.000,E1 192.647} C_DIS
LIN {X 0.114,Y -447.578,Z 1075.865,A 0.000,B 0.000,C 90.000,E1 191.658} C_DIS
LIN {X -0.080,Y -460.812,Z 1075.851,A 0.000,B 0.000,C 90.000,E1 189.265} C_DIS
LIN {X -0.063,Y -468.029,Z 1075.844,A 0.000,B 0.000,C 90.000,E1 187.992} C_DIS
LIN {X -0.048,Y -474.301,Z 1075.838,A 0.000,B 0.000,C 90.000,E1 186.891} C_DIS
LIN {X -0.143,Y -479.422,Z 1075.833,A 0.000,B 0.000,C 90.000,E1 185.967} C_DIS
LIN {X -0.083,Y -485.160,Z 1075.827,A 0.000,B 0.000,C 90.000,E1 184.878} C_DIS
LIN {X 0.102,Y -490.946,Z 1075.821,A 0.000,B 0.000,C 90.000,E1 183.784} C_DIS
LIN {X 0.009,Y -497.331,Z 1075.814,A 0.000,B 0.000,C 90.000,E1 182.579} C_DIS
LIN {X -0.182,Y -502.893,Z 1075.808,A 0.000,B 0.000,C 90.000,E1 181.547} C_DIS
LIN {X -0.013,Y -507.552,Z 1075.804,A 0.000,B 0.000,C 90.000,E1 180.630} C_DIS
LIN {X 0.054,Y -515.273,Z 1075.795,A 0.000,B 0.000,C 90.000,E1 179.141} C_DIS
LIN {X 0.098,Y -520.657,Z 1075.790,A 0.000,B 0.000,C 90.000,E1 178.108} C_DIS
LIN {X 0.120,Y -530.403,Z 1075.779,A 0.000,B 0.000,C 90.000,E1 176.216} C_DIS
LIN {X -0.094,Y -540.059,Z 1075.769,A 0.000,B 0.000,C 90.000,E1 174.375} C_DIS
LIN {X -0.115,Y -548.062,Z 1075.760,A 0.000,B 0.000,C 90.000,E1 172.818} C_DIS
LIN {X -0.026,Y -554.505,Z 1075.753,A 0.000,B 0.000,C 90.000,E1 171.546} C_DIS
LIN {X 0.162,Y -560.850,Z 1075.746,A 0.000,B 0.000,C 90.000,E1 170.274} C_DIS
LIN {X 0.161,Y -568.306,Z 1075.738,A 0.000,B 0.000,C 90.000,E1 168.757} C_DIS
LIN {X -0.214,Y -573.443,Z 1075.732,A 0.000,B 0.000,C 90.000,E1 167.701} C_DIS
LIN {X -0.091,Y -580.904,Z 1075.723,A 0.000,B 0.000,C 90.000,E1 166.061} C_DIS
LIN {X 0.076,Y -585.054,Z 1075.717,A 0.000,B 0.000,C 90.000,E1 165.102} C_DIS
LIN {X 0.067,Y -589.482,Z 1075.711,A 0.000,B 0.000,C 90.000,E1 164.031} C_DIS
LIN {X -0.314,Y -592.709,Z 1075.707,A 0.000,B 0.000,C 90.000,E1 163.268} C_DIS
LIN {X 0.248,Y -595.762,Z 1075.703,A 0.000,B 0.000,C 90.000,E1 162.417} C_DIS
LIN {X -0.197,Y -599.669,Z 1075.697,A 0.000,B 0.000,C 90.000,E1 161.402} C_DIS
LIN {X 0.161,Y -603.295,Z 1075.691,A 0.000,B 0.000,C 90.000,E1 160.315} C_DIS
LIN {X 0.212,Y -606.757,Z 1075.685,A 0.000,B 0.000,C 90.000,E1 159.263} C_DIS
LIN {X 0.044,Y -610.766,Z 1075.678,A 0.000,B 0.000,C 90.000,E1 157.975} C_DIS
LIN {X 0.244,Y -613.159,Z 1075.673,A 0.000,B 0.000,C 90.000,E1 157.177} C_DIS
LIN {X -0.154,Y -616.772,Z 1075.666,A 0.000,B 0.000,C 90.000,E1 155.921} C_DIS
LIN {X 0.055,Y -620.886,Z 1075.658,A 0.000,B 0.000,C 90.000,E1 154.357} C_DIS
LIN {X 0.046,Y -624.066,Z 1075.651,A 0.000,B 0.000,C 90.000,E1 153.076} C_DIS
LIN {X -0.171,Y -627.218,Z 1075.643,A 0.000,B 0.000,C 90.000,E1 151.820} C_DIS
LIN {X -0.099,Y -629.624,Z 1075.638,A 0.000,B 0.000,C 90.000,E1 150.795} C_DIS
LIN {X -0.186,Y -633.052,Z 1075.629,A 0.000,B 0.000,C 90.000,E1 149.282} C_DIS
LIN {X -0.051,Y -636.863,Z 1075.620,A 0.000,B 0.000,C 90.000,E1 147.502} C_DIS
LIN {X 0.189,Y -640.476,Z 1075.610,A 0.000,B 0.000,C 90.000,E1 145.722} C_DIS
LIN {X -0.063,Y -643.478,Z 1075.601,A 0.000,B 0.000,C 90.000,E1 144.242} C_DIS
LIN {X -0.261,Y -646.398,Z 1075.593,A 0.000,B 0.000,C 90.000,E1 142.763} C_DIS
LIN {X 0.026,Y -648.402,Z 1075.588,A 0.000,B 0.000,C 90.000,E1 141.743} C_DIS
LIN {X 0.341,Y -650.376,Z 1075.582,A 0.000,B 0.000,C 90.000,E1 140.723} C_DIS
LIN {X 0.089,Y -653.851,Z 1075.572,A 0.000,B 0.000,C 90.000,E1 139.013} C_DIS
LIN {X -0.115,Y -656.959,Z 1075.564,A 0.000,B 0.000,C 90.000,E1 137.553} C_DIS
LIN {X 0.127,Y -661.781,Z 1075.552,A 0.000,B 0.000,C 90.000,E1 135.324} C_DIS
LIN {X 0.057,Y -665.382,Z 1075.544,A 0.000,B 0.000,C 90.000,E1 133.866} C_DIS
LIN {X 0.083,Y -669.118,Z 1075.536,A 0.000,B 0.000,C 90.000,E1 132.405} C_DIS
LIN {X -0.316,Y -672.891,Z 1075.528,A 0.000,B 0.000,C 90.000,E1 130.987} C_DIS
LIN {X -0.068,Y -676.636,Z 1075.520,A 0.000,B 0.000,C 90.000,E1 129.519} C_DIS
LIN {X -0.103,Y -681.518,Z 1075.509,A 0.000,B 0.000,C 90.000,E1 127.604} C_DIS
LIN {X 0.099,Y -683.399,Z 1075.505,A 0.000,B 0.000,C 90.000,E1 126.870} C_DIS
LIN {X 0.112,Y -686.461,Z 1075.498,A 0.000,B 0.000,C 90.000,E1 125.678} C_DIS
LIN {X 0.178,Y -689.308,Z 1075.492,A 0.000,B 0.000,C 90.000,E1 124.485} C_DIS
LIN {X -0.074,Y -692.810,Z 1075.484,A 0.000,B 0.000,C 90.000,E1 123.086} C_DIS
LIN {X 0.286,Y -695.640,Z 1075.477,A 0.000,B 0.000,C 90.000,E1 121.878} C_DIS
LIN {X 0.099,Y -698.299,Z 1075.471,A 0.000,B 0.000,C 90.000,E1 120.718} C_DIS
LIN {X 0.271,Y -699.768,Z 1075.467,A 0.000,B 0.000,C 90.000,E1 120.001} C_DIS
LIN {X 0.120,Y -701.128,Z 1075.462,A 0.000,B 0.000,C 90.000,E1 119.077} C_DIS
LIN {X 0.050,Y -701.659,Z 1075.459,A 0.000,B 0.000,C 90.000,E1 118.615} C_DIS
LIN {X 0.086,Y -703.473,Z 1075.449,A 0.000,B 0.000,C 90.000,E1 116.744} C_DIS
LIN {X -0.065,Y -704.580,Z 1075.442,A 0.000,B 0.000,C 90.000,E1 115.591} C_DIS
LIN {X -0.430,Y -704.908,Z 1075.440,A 0.000,B 0.000,C 90.000,E1 115.155} C_DIS
LIN {X 0.144,Y -705.057,Z 1075.437,A 0.000,B 0.000,C 90.000,E1 114.643} C_DIS
LIN {X -0.215,Y -704.615,Z 1075.434,A 0.000,B 0.000,C 90.000,E1 114.207} C_DIS
LIN {X 0.070,Y -704.281,Z 1075.433,A 0.000,B 0.000,C 90.000,E1 113.951} C_DIS
LIN {X -0.291,Y -702.736,Z 1075.431,A 0.000,B 0.000,C 90.000,E1 113.515} C_DIS
LIN {X -0.013,Y -701.623,Z 1075.429,A 0.000,B 0.000,C 90.000,E1 113.259} C_DIS
LIN {X 0.254,Y -698.026,Z 1075.427,A 0.000,B 0.000,C 90.000,E1 112.770} C_DIS
LIN {X 0.384,Y -696.862,Z 1075.426,A 0.000,B 0.000,C 90.000,E1 112.642} C_DIS
LIN {X -0.130,Y -695.064,Z 1075.425,A 0.000,B 0.000,C 90.000,E1 112.567} C_DIS
LIN {X 0.188,Y -687.693,Z 1075.423,A 0.000,B 0.000,C 90.000,E1 112.206} C_DIS
LIN {X -0.050,Y -685.671,Z 1075.423,A 0.000,B 0.000,C 90.000,E1 112.153} C_DIS
LIN {X 0.150,Y -684.076,Z 1075.423,A 0.000,B 0.000,C 90.000,E1 112.099} C_DIS
LIN {X -0.080,Y -676.724,Z 1075.422,A 0.000,B 0.000,C 90.000,E1 112.025} C_DIS
LIN {X -0.186,Y -675.407,Z 1075.422,A 0.000,B 0.000,C 90.000,E1 112.025} C_DIS
LIN {X -0.214,Y -606.598,Z 1075.422,A 0.000,B 0.000,C 90.000,E1 112.025} C_DIS
LIN {X 0.057,Y -601.413,Z 1075.421,A 0.000,B 0.000,C 90.000,E1 111.770} C_DIS
LIN {X 0.152,Y -596.904,Z 1075.419,A 0.000,B 0.000,C 90.000,E1 111.482} C_DIS
LIN {X -0.125,Y -591.457,Z 1075.417,A 0.000,B 0.000,C 90.000,E1 111.099} C_DIS
LIN {X 0.201,Y -582.225,Z 1075.413,A 0.000,B 0.000,C 90.000,E1 110.301} C_DIS
LIN {X -0.071,Y -575.491,Z 1075.410,A 0.000,B 0.000,C 90.000,E1 109.758} C_DIS
LIN {X 0.289,Y -569.330,Z 1075.407,A 0.000,B 0.000,C 90.000,E1 109.268} C_DIS
LIN {X 0.207,Y -561.421,Z 1075.405,A 0.000,B 0.000,C 90.000,E1 108.779} C_DIS
LIN {X 0.168,Y -554.811,Z 1075.402,A 0.000,B 0.000,C 90.000,E1 108.417} C_DIS
LIN {X -0.049,Y -549.270,Z 1075.400,A 0.000,B 0.000,C 90.000,E1 108.055} C_DIS
LIN {X -0.125,Y -547.721,Z 1075.399,A 0.000,B 0.000,C 90.000,E1 107.873} C_DIS
LIN {X -0.166,Y -547.689,Z 1075.399,A 0.000,B 0.000,C 90.000,E1 107.873} C_DIS
LIN {X -0.079,Y -547.313,Z 1075.398,A 0.000,B 0.000,C 90.000,E1 107.583} C_DIS
LIN {X 0.119,Y -547.594,Z 1075.394,A 0.000,B 0.000,C 90.000,E1 106.858} C_DIS
LIN {X 0.115,Y -548.380,Z 1075.388,A 0.000,B 0.000,C 90.000,E1 105.733} C_DIS
LIN {X 0.156,Y -549.961,Z 1075.375,A 0.000,B 0.000,C 90.000,E1 103.480} C_DIS
LIN {X -0.015,Y -551.620,Z 1075.364,A 0.000,B 0.000,C 90.000,E1 101.535} C_DIS
LIN {X -0.254,Y -553.915,Z 1075.352,A 0.000,B 0.000,C 90.000,E1 99.321} C_DIS
LIN {X -0.100,Y -556.094,Z 1075.341,A 0.000,B 0.000,C 90.000,E1 97.352} C_DIS
LIN {X -0.158,Y -557.624,Z 1075.333,A 0.000,B 0.000,C 90.000,E1 95.967} C_DIS
LIN {X -0.248,Y -559.031,Z 1075.325,A 0.000,B 0.000,C 90.000,E1 94.588} C_DIS
LIN {X 0.211,Y -559.921,Z 1075.318,A 0.000,B 0.000,C 90.000,E1 93.154} C_DIS
LIN {X 0.154,Y -560.663,Z 1075.310,A 0.000,B 0.000,C 90.000,E1 91.776} C_DIS
LIN {X 0.165,Y -561.482,Z 1075.301,A 0.000,B 0.000,C 90.000,E1 90.115} C_DIS
LIN {X -0.269,Y -562.176,Z 1075.290,A 0.000,B 0.000,C 90.000,E1 88.224} C_DIS
LIN {X 0.274,Y -562.717,Z 1075.282,A 0.000,B 0.000,C 90.000,E1 86.788} C_DIS
LIN {X 0.239,Y -563.265,Z 1075.275,A 0.000,B 0.000,C 90.000,E1 85.412} C_DIS
LIN {X -0.165,Y -563.805,Z 1075.266,A 0.000,B 0.000,C 90.000,E1 83.799} C_DIS
LIN {X 0.158,Y -564.384,Z 1075.255,A 0.000,B 0.000,C 90.000,E1 81.837} C_DIS
LIN {X 0.001,Y -564.556,Z 1075.250,A 0.000,B 0.000,C 90.000,E1 81.027} C_DIS
LIN {X 0.172,Y -565.128,Z 1075.243,A 0.000,B 0.000,C 90.000,E1 79.634} C_DIS
LIN {X -0.096,Y -565.762,Z 1075.235,A 0.000,B 0.000,C 90.000,E1 78.285} C_DIS
LIN {X -0.077,Y -567.061,Z 1075.221,A 0.000,B 0.000,C 90.000,E1 75.811} C_DIS
LIN {X 0.077,Y -569.194,Z 1075.204,A 0.000,B 0.000,C 90.000,E1 72.779} C_DIS
LIN {X -0.023,Y -570.520,Z 1075.195,A 0.000,B 0.000,C 90.000,E1 71.148} C_DIS
LIN {X 0.253,Y -572.129,Z 1075.185,A 0.000,B 0.000,C 90.000,E1 69.209} C_DIS
LIN {X -0.308,Y -573.688,Z 1075.174,A 0.000,B 0.000,C 90.000,E1 67.358} C_DIS
LIN {X 0.305,Y -574.981,Z 1075.165,A 0.000,B 0.000,C 90.000,E1 65.665} C_DIS
LIN {X 0.057,Y -575.867,Z 1075.157,A 0.000,B 0.000,C 90.000,E1 64.332} C_DIS
LIN {X -0.180,Y -576.643,Z 1075.150,A 0.000,B 0.000,C 90.000,E1 62.999} C_DIS
LIN {X 0.002,Y -577.256,Z 1075.144,A 0.000,B 0.000,C 90.000,E1 61.897} C_DIS
LIN {X 0.042,Y -578.051,Z 1075.136,A 0.000,B 0.000,C 90.000,E1 60.539} C_DIS
LIN {X 0.025,Y -578.591,Z 1075.130,A 0.000,B 0.000,C 90.000,E1 59.459} C_DIS
LIN {X -0.279,Y -579.336,Z 1075.121,A 0.000,B 0.000,C 90.000,E1 57.867} C_DIS
LIN {X 0.047,Y -580.102,Z 1075.112,A 0.000,B 0.000,C 90.000,E1 56.215} C_DIS
LIN {X -0.085,Y -580.744,Z 1075.103,A 0.000,B 0.000,C 90.000,E1 54.609} C_DIS
LIN {X -0.037,Y -581.082,Z 1075.096,A 0.000,B 0.000,C 90.000,E1 53.256} C_DIS
LIN {X 0.127,Y -581.251,Z 1075.091,A 0.000,B 0.000,C 90.000,E1 52.431} C_DIS
LIN {X 0.183,Y -581.253,Z 1075.087,A 0.000,B 0.000,C 90.000,E1 51.618} C_DIS
LIN {X -0.037,Y -581.046,Z 1075.081,A 0.000,B 0.000,C 90.000,E1 50.561} C_DIS
LIN {X -0.086,Y -580.650,Z 1075.073,A 0.000,B 0.000,C 90.000,E1 49.218} C_DIS
LIN {X -0.310,Y -580.209,Z 1075.068,A 0.000,B 0.000,C 90.000,E1 48.162} C_DIS
LIN {X -0.003,Y -579.499,Z 1075.060,A 0.000,B 0.000,C 90.000,E1 46.782} C_DIS
LIN {X -0.281,Y -578.776,Z 1075.054,A 0.000,B 0.000,C 90.000,E1 45.729} C_DIS
LIN {X 0.257,Y -577.833,Z 1075.048,A 0.000,B 0.000,C 90.000,E1 44.595} C_DIS
LIN {X -0.041,Y -576.607,Z 1075.042,A 0.000,B 0.000,C 90.000,E1 43.542} C_DIS
LIN {X 0.197,Y -574.741,Z 1075.034,A 0.000,B 0.000,C 90.000,E1 42.162} C_DIS
LIN {X -0.244,Y -573.548,Z 1075.030,A 0.000,B 0.000,C 90.000,E1 41.391} C_DIS
LIN {X -0.061,Y -570.985,Z 1075.022,A 0.000,B 0.000,C 90.000,E1 40.011} C_DIS
LIN {X 0.018,Y -568.525,Z 1075.016,A 0.000,B 0.000,C 90.000,E1 38.910} C_DIS
LIN {X -0.055,Y -566.507,Z 1075.012,A 0.000,B 0.000,C 90.000,E1 38.096} C_DIS
LIN {X -0.153,Y -564.230,Z 1075.007,A 0.000,B 0.000,C 90.000,E1 37.282} C_DIS
